// Mitsubishi GX Works2 project: wakom   PLC: Q02/Q02H

TYPE QD75_POS : STRUCT
  id : INT;
  mcode : INT;
  dwell_time : INT;
  spare : INT;
  speed : DINT;
  address : DINT;
  arc_address : DINT;
END_STRUCT END_TYPE

TYPE CAR_DATA : STRUCT
  cid : INT;
  enter_time : ARRAY [0..6] OF INT;
  leave_time : ARRAY [0..6] OF INT;
  proc_time : ARRAY [0..6] OF INT;
END_STRUCT END_TYPE

TYPE TK_POS : STRUCT
  h_lock : DINT;
  h_unlock : DINT;
  v_bottom : DINT;
  h_lock2 : DINT;
  h_unlock2 : DINT;
  v_bottom2 : DINT;
END_STRUCT END_TYPE

TYPE TK_CNF : STRUCT
  take_weight : INT;
  next_tank : ARRAY [0..4] OF INT;
  is_bypass : INT;
END_STRUCT END_TYPE

TYPE RECIPE : STRUCT
  tk_data : ARRAY [0..249] OF INT;
  sys_data : INT;
END_STRUCT END_TYPE

TYPE TK_STATUS : STRUCT
  permit_put : BOOL;
  cover_is_open : BOOL;
  cmd_open_cover : BOOL;
  cmd_close_cover : BOOL;
  permit_take : BOOL;
  rb_inter_lock : INT;
  pc_key : INT;
END_STRUCT END_TYPE

TYPE RB_STATUS : STRUCT
  pc_tid : INT;
  pc_key : INT;
  h_cur_pos : DINT;
  v_cur_pos : DINT;
  v_error_code : INT;
  v_alarm_code : INT;
  v_serve_alarm_code : INT;
  v_action_status : INT;
  v_status : INT;
  rb_state : INT;
  target_tid : INT;
  cur_tid : INT;
  from_tid : INT;
  to_tid : INT;
  v_xy : INT;
  v_cur_speed : DINT;
  v_bit : INT;
  h_cur_speed : DINT;
  h_error_code : INT;
  h_alarm_code : INT;
  h_serve_alarm_code : INT;
  h_action_status : INT;
  h_status : INT;
  h_xy : INT;
  h_bit : INT;
  h_address : DINT;
  h_speed : DINT;
  v_address : DINT;
  v_speed : DINT;
  rb_bit : INT;
END_STRUCT END_TYPE

TYPE SYS_STATUS : STRUCT
  amode : BOOL;
  mmode : BOOL;
  cycle_stop : BOOL;
  enable_run : BOOL;
  key_reset : BOOL;
  rcpid : INT;
END_STRUCT END_TYPE

TYPE ALARM : STRUCT
  tk : ARRAY [0..6] OF DINT;
  rb : ARRAY [0..0] OF DINT;
  emo : BOOL;
  leak : BOOL;
END_STRUCT END_TYPE

TYPE DIW_RCP : STRUCT
  LoopCount : INT;
  uiRemain : ARRAY [0..5] OF INT;
  uiCmd : ARRAY [0..5] OF INT;
  spare : ARRAY [0..36] OF INT;
END_STRUCT END_TYPE

// global labels: Global1
VAR_GLOBAL
  g_tk_status : ARRAY [0..6] OF TK_STATUS;
  g_rb_status : ARRAY [0..0] OF RB_STATUS;
  g_pc_cmd AT D900 : ARRAY [0..99] OF INT;
  g_recipe : RECIPE;
  g_tk_cnf : ARRAY [0..6] OF TK_CNF;
  g_tk_pos : ARRAY [0..6] OF TK_POS;
END_VAR
VAR_GLOBAL CONSTANT
  g_safe_height : DINT;
END_VAR
VAR_GLOBAL
  g_tk_car : ARRAY [0..6] OF CAR_DATA;
  g_rb_car : ARRAY [0..0] OF CAR_DATA;
  g_sys_status : SYS_STATUS;
  g_alarm : ALARM;
END_VAR
VAR_GLOBAL CONSTANT
  g_rcp_max_size : INT := 50;
END_VAR

// task task01 (event TRUE, interval 0, priority 31): robot01
// task task02 (event TRUE, interval 0, priority 31): main

PROGRAM robot01
VAR
  axis_h : rb_axis;
  axis_v : rb_axis;
  rb_dispatch_1 : rb_dispatch;
END_VAR
(* structured ladder/FBD written out as ST: instructions are called as NAME(EN, inputs, outputs); _pN, _eN, _tN stand for wires *)
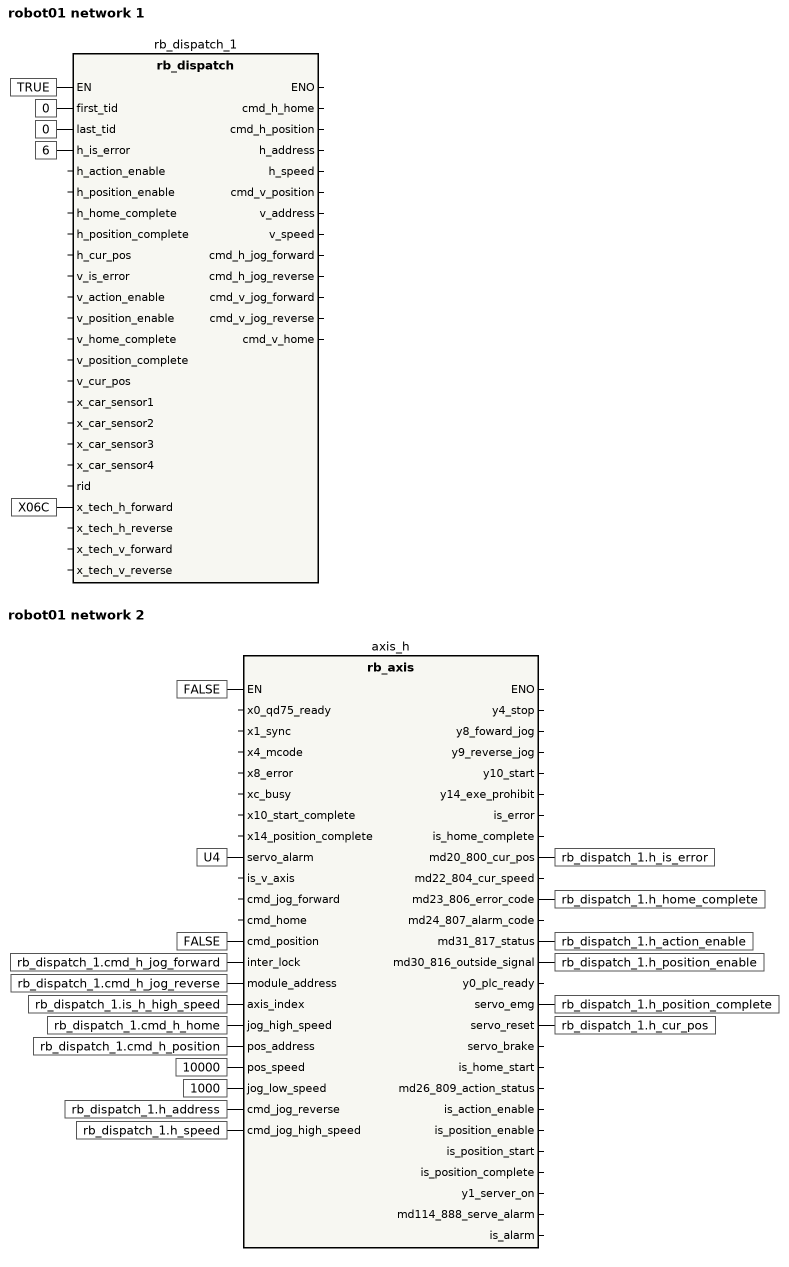
(* network 1 *)
rb_dispatch_1(EN := TRUE, first_tid := 0, last_tid := 0, h_is_error := 6, x_tech_h_forward := X06C);
(* network 2 *)
axis_h(EN := FALSE, servo_alarm := U4, cmd_position := FALSE, inter_lock := rb_dispatch_1.cmd_h_jog_forward, module_address := rb_dispatch_1.cmd_h_jog_reverse, axis_index := rb_dispatch_1.is_h_high_speed, jog_high_speed := rb_dispatch_1.cmd_h_home, pos_address := rb_dispatch_1.cmd_h_position, pos_speed := 10000, jog_low_speed := 1000, cmd_jog_reverse := rb_dispatch_1.h_address, cmd_jog_high_speed := rb_dispatch_1.h_speed, md20_800_cur_pos => rb_dispatch_1.h_is_error, md23_806_error_code => rb_dispatch_1.h_home_complete, md31_817_status => rb_dispatch_1.h_action_enable, md30_816_outside_signal => rb_dispatch_1.h_position_enable, servo_emg => rb_dispatch_1.h_position_complete, servo_reset => rb_dispatch_1.h_cur_pos);
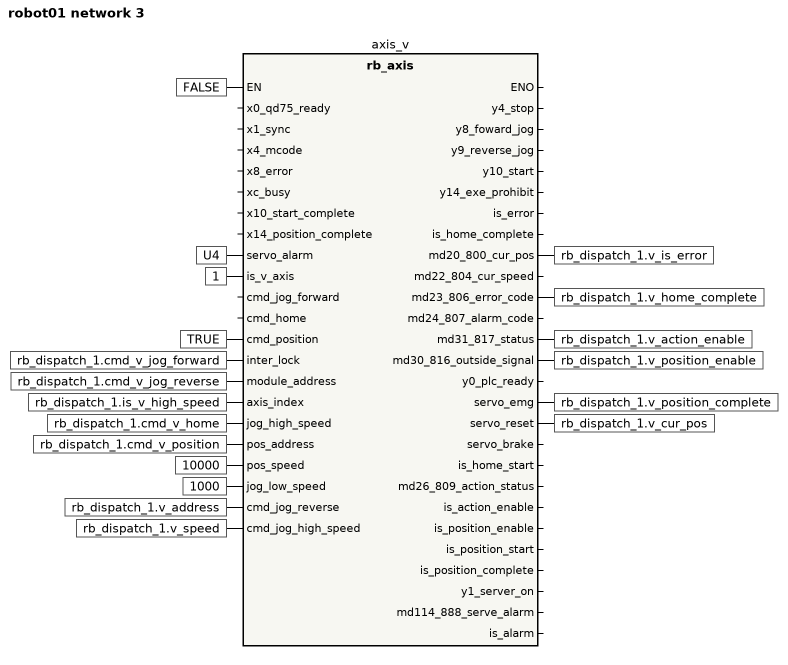
(* network 3 *)
axis_v(EN := FALSE, servo_alarm := U4, is_v_axis := 1, cmd_position := TRUE, inter_lock := rb_dispatch_1.cmd_v_jog_forward, module_address := rb_dispatch_1.cmd_v_jog_reverse, axis_index := rb_dispatch_1.is_v_high_speed, jog_high_speed := rb_dispatch_1.cmd_v_home, pos_address := rb_dispatch_1.cmd_v_position, pos_speed := 10000, jog_low_speed := 1000, cmd_jog_reverse := rb_dispatch_1.v_address, cmd_jog_high_speed := rb_dispatch_1.v_speed, md20_800_cur_pos => rb_dispatch_1.v_is_error, md23_806_error_code => rb_dispatch_1.v_home_complete, md31_817_status => rb_dispatch_1.v_action_enable, md30_816_outside_signal => rb_dispatch_1.v_position_enable, servo_emg => rb_dispatch_1.v_position_complete, servo_reset => rb_dispatch_1.v_cur_pos);
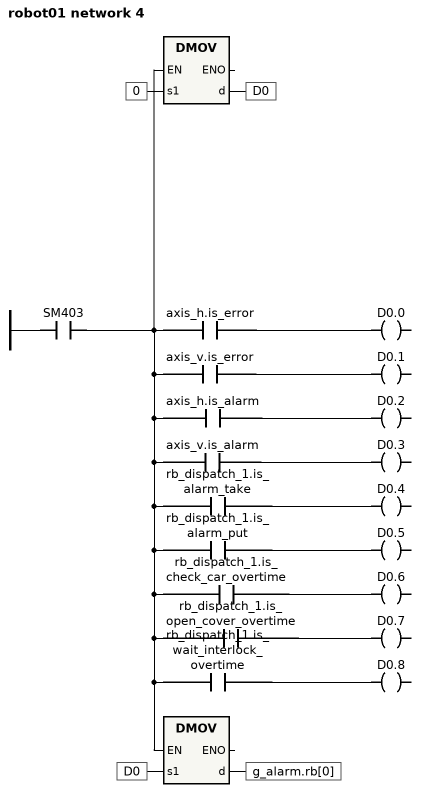
(* network 4 *)
DMOV(SM403, 0, D0);
D0.0 := SM403 AND axis_h.is_error;
D0.1 := SM403 AND axis_v.is_error;
D0.2 := SM403 AND axis_h.is_alarm;
D0.3 := SM403 AND axis_v.is_alarm;
D0.4 := SM403 AND rb_dispatch_1.is_alarm_take;
D0.5 := SM403 AND rb_dispatch_1.is_alarm_put;
D0.6 := SM403 AND rb_dispatch_1.is_check_car_overtime;
D0.7 := SM403 AND rb_dispatch_1.is_open_cover_overtime;
D0.8 := SM403 AND rb_dispatch_1.is_wait_interlock_overtime;
DMOV(SM403, D0, g_alarm.rb[0]);
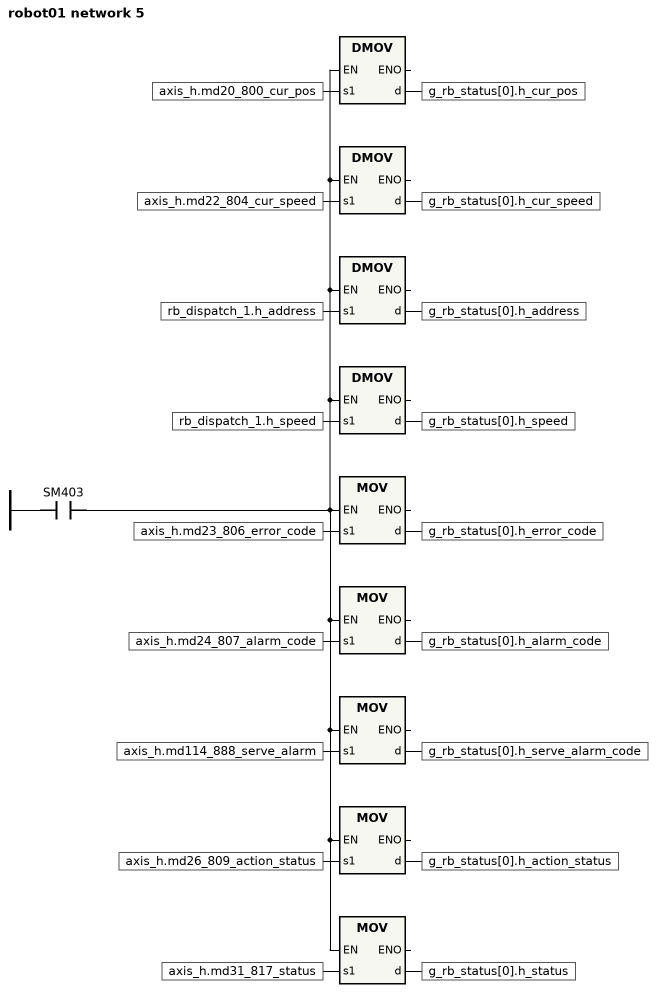
(* network 5 *)
DMOV(SM403, axis_h.md20_800_cur_pos, g_rb_status[0].h_cur_pos);
DMOV(SM403, axis_h.md22_804_cur_speed, g_rb_status[0].h_cur_speed);
DMOV(SM403, rb_dispatch_1.h_address, g_rb_status[0].h_address);
DMOV(SM403, rb_dispatch_1.h_speed, g_rb_status[0].h_speed);
MOV(SM403, axis_h.md23_806_error_code, g_rb_status[0].h_error_code);
MOV(SM403, axis_h.md24_807_alarm_code, g_rb_status[0].h_alarm_code);
MOV(SM403, axis_h.md114_888_serve_alarm, g_rb_status[0].h_serve_alarm_code);
MOV(SM403, axis_h.md26_809_action_status, g_rb_status[0].h_action_status);
MOV(SM403, axis_h.md31_817_status, g_rb_status[0].h_status);
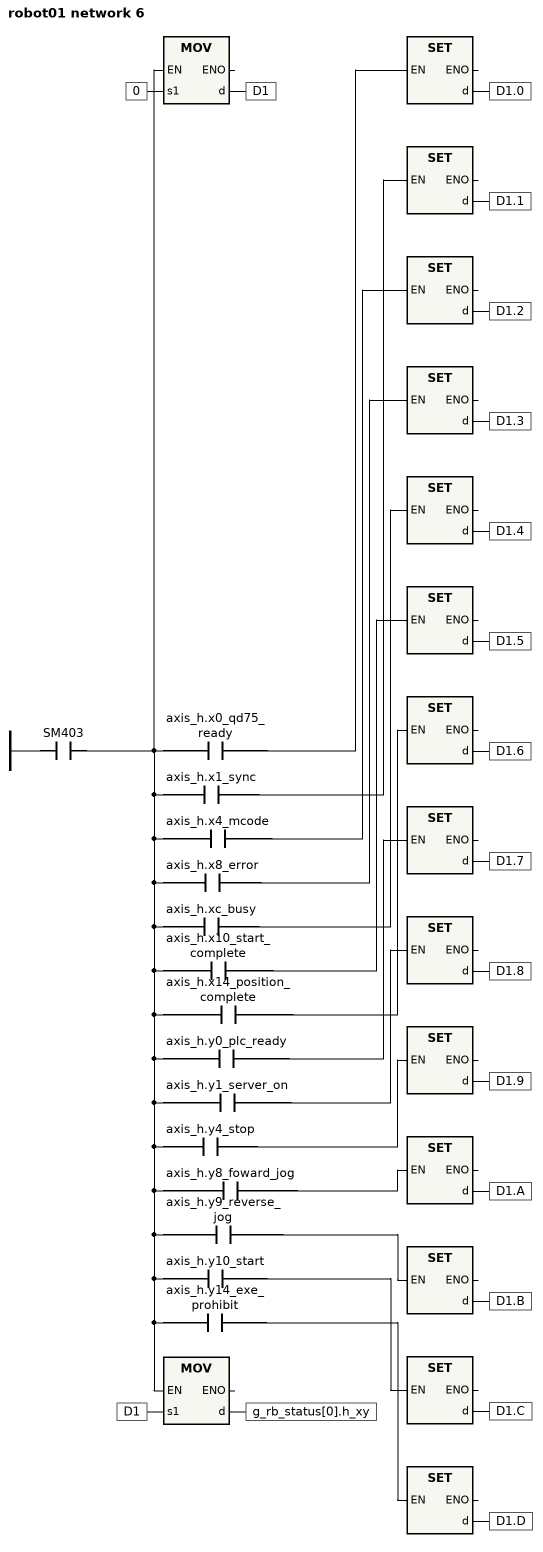
(* network 6 *)
MOV(SM403, 0, D1);
SET(SM403 AND axis_h.x0_qd75_ready, D1.0);
SET(SM403 AND axis_h.x1_sync, D1.1);
SET(SM403 AND axis_h.x4_mcode, D1.2);
SET(SM403 AND axis_h.x8_error, D1.3);
SET(SM403 AND axis_h.xc_busy, D1.4);
SET(SM403 AND axis_h.x10_start_complete, D1.5);
SET(SM403 AND axis_h.x14_position_complete, D1.6);
SET(SM403 AND axis_h.y0_plc_ready, D1.7);
SET(SM403 AND axis_h.y1_server_on, D1.8);
SET(SM403 AND axis_h.y4_stop, D1.9);
SET(SM403 AND axis_h.y8_foward_jog, D1.A);
SET(SM403 AND axis_h.y9_reverse_jog, D1.B);
SET(SM403 AND axis_h.y10_start, D1.C);
SET(SM403 AND axis_h.y14_exe_prohibit, D1.D);
MOV(SM403, D1, g_rb_status[0].h_xy);
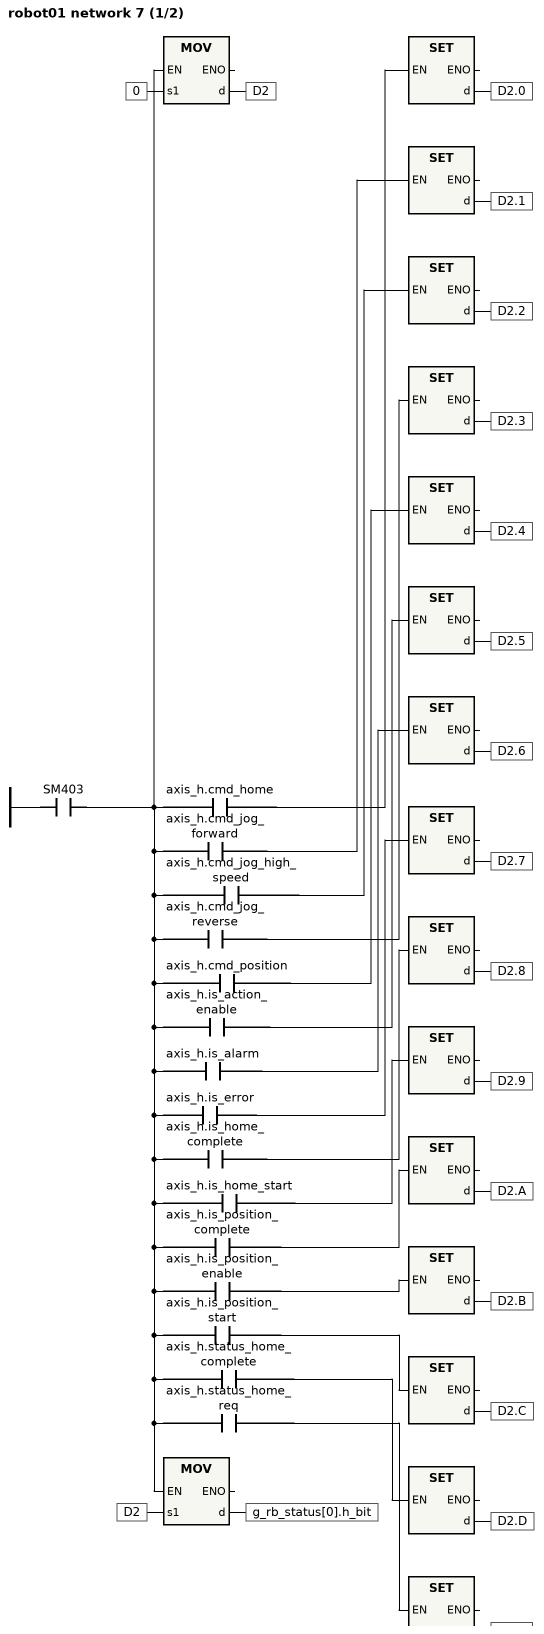
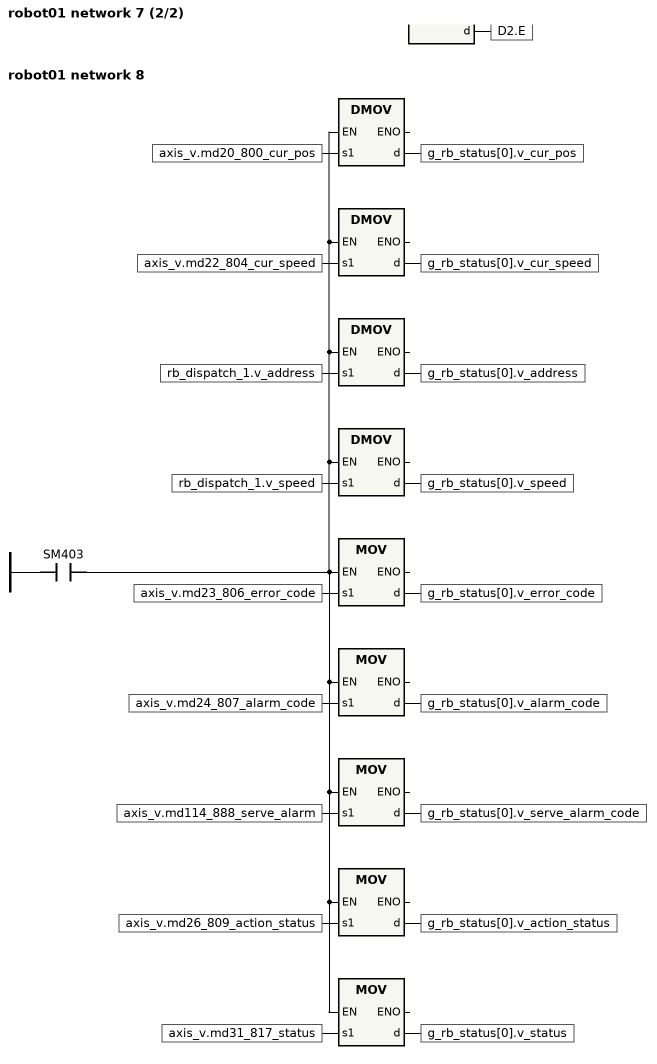
(* network 7 *)
MOV(SM403, 0, D2);
SET(SM403 AND axis_h.cmd_home, D2.0);
SET(SM403 AND axis_h.cmd_jog_forward, D2.1);
SET(SM403 AND axis_h.cmd_jog_high_speed, D2.2);
SET(SM403 AND axis_h.cmd_jog_reverse, D2.3);
SET(SM403 AND axis_h.cmd_position, D2.4);
SET(SM403 AND axis_h.is_action_enable, D2.5);
SET(SM403 AND axis_h.is_alarm, D2.6);
SET(SM403 AND axis_h.is_error, D2.7);
SET(SM403 AND axis_h.is_home_complete, D2.8);
SET(SM403 AND axis_h.is_home_start, D2.9);
SET(SM403 AND axis_h.is_position_complete, D2.A);
SET(SM403 AND axis_h.is_position_enable, D2.B);
SET(SM403 AND axis_h.is_position_start, D2.C);
SET(SM403 AND axis_h.status_home_complete, D2.D);
SET(SM403 AND axis_h.status_home_req, D2.E);
MOV(SM403, D2, g_rb_status[0].h_bit);
(* network 8 *)
DMOV(SM403, axis_v.md20_800_cur_pos, g_rb_status[0].v_cur_pos);
DMOV(SM403, axis_v.md22_804_cur_speed, g_rb_status[0].v_cur_speed);
DMOV(SM403, rb_dispatch_1.v_address, g_rb_status[0].v_address);
DMOV(SM403, rb_dispatch_1.v_speed, g_rb_status[0].v_speed);
MOV(SM403, axis_v.md23_806_error_code, g_rb_status[0].v_error_code);
MOV(SM403, axis_v.md24_807_alarm_code, g_rb_status[0].v_alarm_code);
MOV(SM403, axis_v.md114_888_serve_alarm, g_rb_status[0].v_serve_alarm_code);
MOV(SM403, axis_v.md26_809_action_status, g_rb_status[0].v_action_status);
MOV(SM403, axis_v.md31_817_status, g_rb_status[0].v_status);
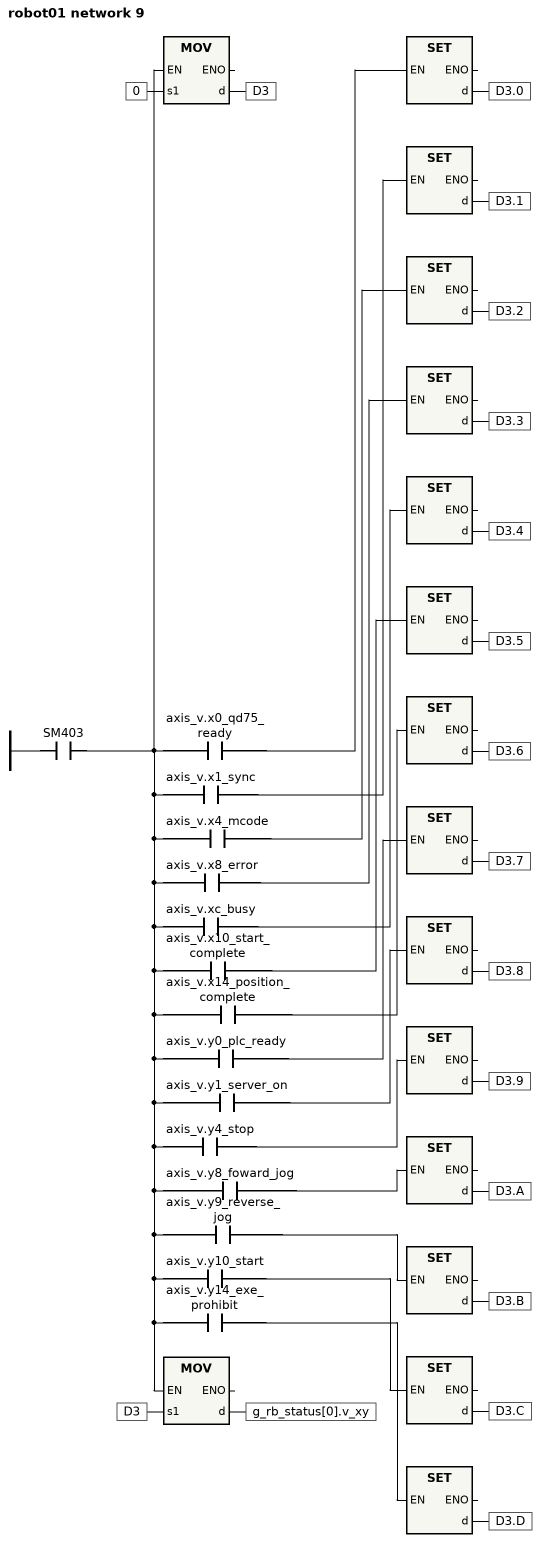
(* network 9 *)
MOV(SM403, 0, D3);
SET(SM403 AND axis_v.x0_qd75_ready, D3.0);
SET(SM403 AND axis_v.x1_sync, D3.1);
SET(SM403 AND axis_v.x4_mcode, D3.2);
SET(SM403 AND axis_v.x8_error, D3.3);
SET(SM403 AND axis_v.xc_busy, D3.4);
SET(SM403 AND axis_v.x10_start_complete, D3.5);
SET(SM403 AND axis_v.x14_position_complete, D3.6);
SET(SM403 AND axis_v.y0_plc_ready, D3.7);
SET(SM403 AND axis_v.y1_server_on, D3.8);
SET(SM403 AND axis_v.y4_stop, D3.9);
SET(SM403 AND axis_v.y8_foward_jog, D3.A);
SET(SM403 AND axis_v.y9_reverse_jog, D3.B);
SET(SM403 AND axis_v.y10_start, D3.C);
SET(SM403 AND axis_v.y14_exe_prohibit, D3.D);
MOV(SM403, D3, g_rb_status[0].v_xy);
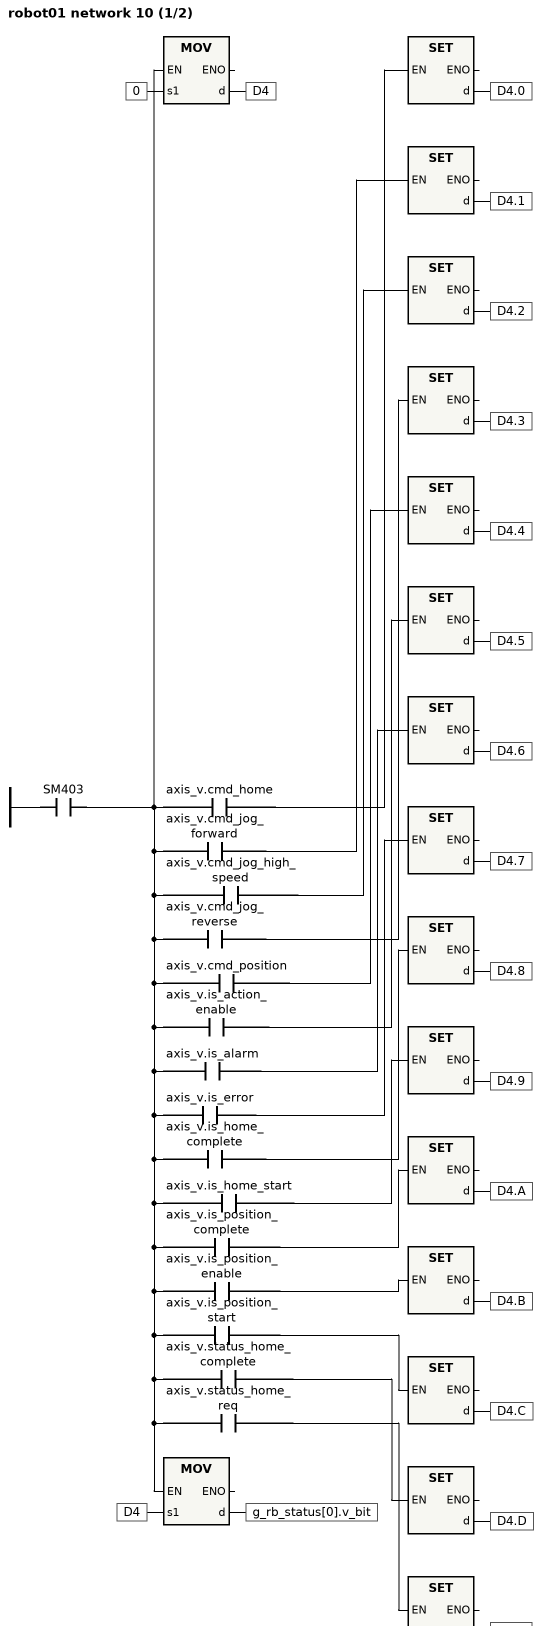
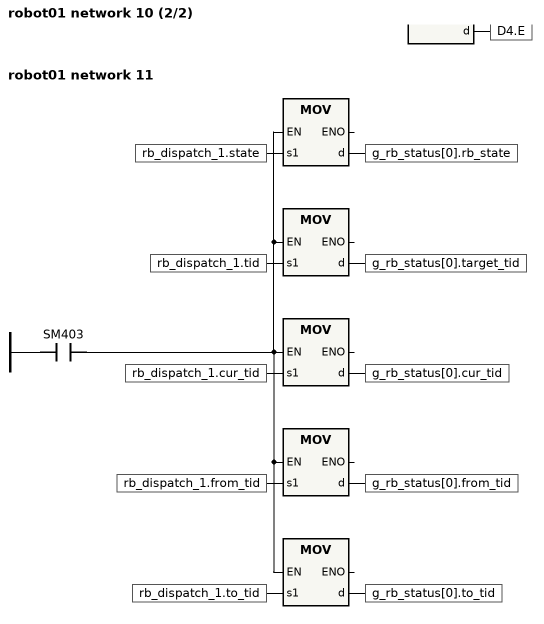
(* network 10 *)
MOV(SM403, 0, D4);
SET(SM403 AND axis_v.cmd_home, D4.0);
SET(SM403 AND axis_v.cmd_jog_forward, D4.1);
SET(SM403 AND axis_v.cmd_jog_high_speed, D4.2);
SET(SM403 AND axis_v.cmd_jog_reverse, D4.3);
SET(SM403 AND axis_v.cmd_position, D4.4);
SET(SM403 AND axis_v.is_action_enable, D4.5);
SET(SM403 AND axis_v.is_alarm, D4.6);
SET(SM403 AND axis_v.is_error, D4.7);
SET(SM403 AND axis_v.is_home_complete, D4.8);
SET(SM403 AND axis_v.is_home_start, D4.9);
SET(SM403 AND axis_v.is_position_complete, D4.A);
SET(SM403 AND axis_v.is_position_enable, D4.B);
SET(SM403 AND axis_v.is_position_start, D4.C);
SET(SM403 AND axis_v.status_home_complete, D4.D);
SET(SM403 AND axis_v.status_home_req, D4.E);
MOV(SM403, D4, g_rb_status[0].v_bit);
(* network 11 *)
MOV(SM403, rb_dispatch_1.state, g_rb_status[0].rb_state);
MOV(SM403, rb_dispatch_1.tid, g_rb_status[0].target_tid);
MOV(SM403, rb_dispatch_1.cur_tid, g_rb_status[0].cur_tid);
MOV(SM403, rb_dispatch_1.from_tid, g_rb_status[0].from_tid);
MOV(SM403, rb_dispatch_1.to_tid, g_rb_status[0].to_tid);
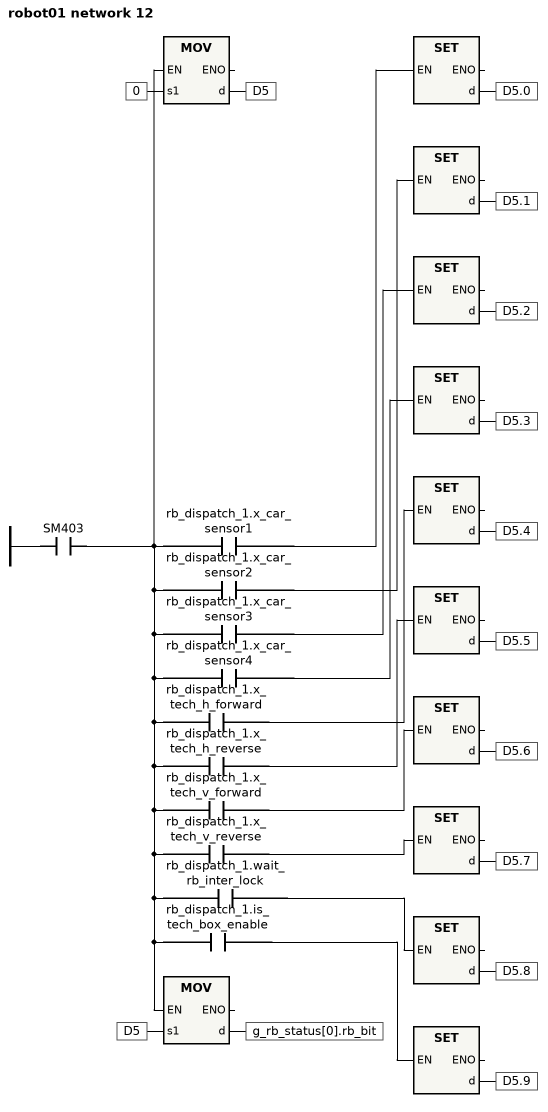
(* network 12 *)
MOV(SM403, 0, D5);
SET(SM403 AND rb_dispatch_1.x_car_sensor1, D5.0);
SET(SM403 AND rb_dispatch_1.x_car_sensor2, D5.1);
SET(SM403 AND rb_dispatch_1.x_car_sensor3, D5.2);
SET(SM403 AND rb_dispatch_1.x_car_sensor4, D5.3);
SET(SM403 AND rb_dispatch_1.x_tech_h_forward, D5.4);
SET(SM403 AND rb_dispatch_1.x_tech_h_reverse, D5.5);
SET(SM403 AND rb_dispatch_1.x_tech_v_forward, D5.6);
SET(SM403 AND rb_dispatch_1.x_tech_v_reverse, D5.7);
SET(SM403 AND rb_dispatch_1.wait_rb_inter_lock, D5.8);
SET(SM403 AND rb_dispatch_1.is_tech_box_enable, D5.9);
MOV(SM403, D5, g_rb_status[0].rb_bit);
END_PROGRAM

FUNCTION_BLOCK rb_axis
VAR_INPUT
  x0_qd75_ready : BOOL;
  x1_sync : BOOL;
  x4_mcode : BOOL;
  x8_error : BOOL;
  xc_busy : BOOL;
  x10_start_complete : BOOL;
END_VAR
VAR_OUTPUT
  y4_stop : BOOL;
  y8_foward_jog : BOOL;
  y9_reverse_jog : BOOL;
  y10_start : BOOL;  (* 定位启动信号 *)
END_VAR
VAR_INPUT
  x14_position_complete : BOOL;
END_VAR
VAR_OUTPUT
  y14_exe_prohibit : BOOL;
  is_error : BOOL;
  is_home_complete : BOOL;
END_VAR
VAR CONSTANT
  cd5_1502_error_reset : INT := 1502;
  cd7_1504_mcode_off : INT := 1504;
END_VAR
VAR_OUTPUT
  md20_800_cur_pos : DINT;
  md22_804_cur_speed : DINT;
  md23_806_error_code : INT;
  md24_807_alarm_code : INT;
  md31_817_status : INT;
  md30_816_outside_signal : WORD;  (* Md.30外部输入输出信号 *)
  y0_plc_ready : BOOL;
  servo_emg : BOOL;
  servo_reset : BOOL;
  servo_brake : BOOL;
END_VAR
VAR_INPUT
  servo_alarm : BOOL;
  is_v_axis : BOOL;
  cmd_jog_forward : BOOL;
END_VAR
VAR CONSTANT
  cd17_1518_jog_speed : INT := 1518;
END_VAR
VAR_INPUT
  cmd_home : BOOL;
END_VAR
VAR_OUTPUT
  is_home_start : BOOL;
END_VAR
VAR_INPUT
  cmd_position : BOOL;
END_VAR
VAR CONSTANT
  cd3_1500_position_num : INT := 1500;
  da2000_position : INT := 2000;
END_VAR
VAR_OUTPUT
  md26_809_action_status : INT;
  is_action_enable : BOOL;
  is_position_enable : BOOL;
  is_position_start : BOOL;
  is_position_complete : BOOL;
END_VAR
VAR_INPUT
  inter_lock : BOOL;
  module_address : INT;
  axis_index : INT;
  jog_high_speed : DINT;
  pos_address : DINT;
END_VAR
VAR
  outside_down_limit : BOOL;
  outside_up_limit : BOOL;
  outside_stop : BOOL;
  status_home_req : BOOL;
  status_home_complete : BOOL;
END_VAR
VAR_INPUT
  pos_speed : DINT;
END_VAR
VAR
  pos_data : QD75_POS;
  home_overtime : BOOL;
  TON_home : TON;
END_VAR
VAR CONSTANT
  TON_home_time : TIME;
END_VAR
VAR
  position_overtime : BOOL;
  TON_position : TON;
END_VAR
VAR CONSTANT
  TON_position_time : TIME;
END_VAR
VAR_INPUT
  jog_low_speed : DINT;
END_VAR
VAR_OUTPUT
  y1_server_on : BOOL;
END_VAR
VAR_INPUT
  cmd_jog_reverse : BOOL;
  cmd_jog_high_speed : BOOL;
END_VAR
VAR_OUTPUT
  md114_888_serve_alarm : INT;
  is_alarm : BOOL;
END_VAR
VAR
  status_alarm : BOOL;
END_VAR
(* structured ladder/FBD written out as ST: instructions are called as NAME(EN, inputs, outputs); _pN, _eN, _tN stand for wires *)
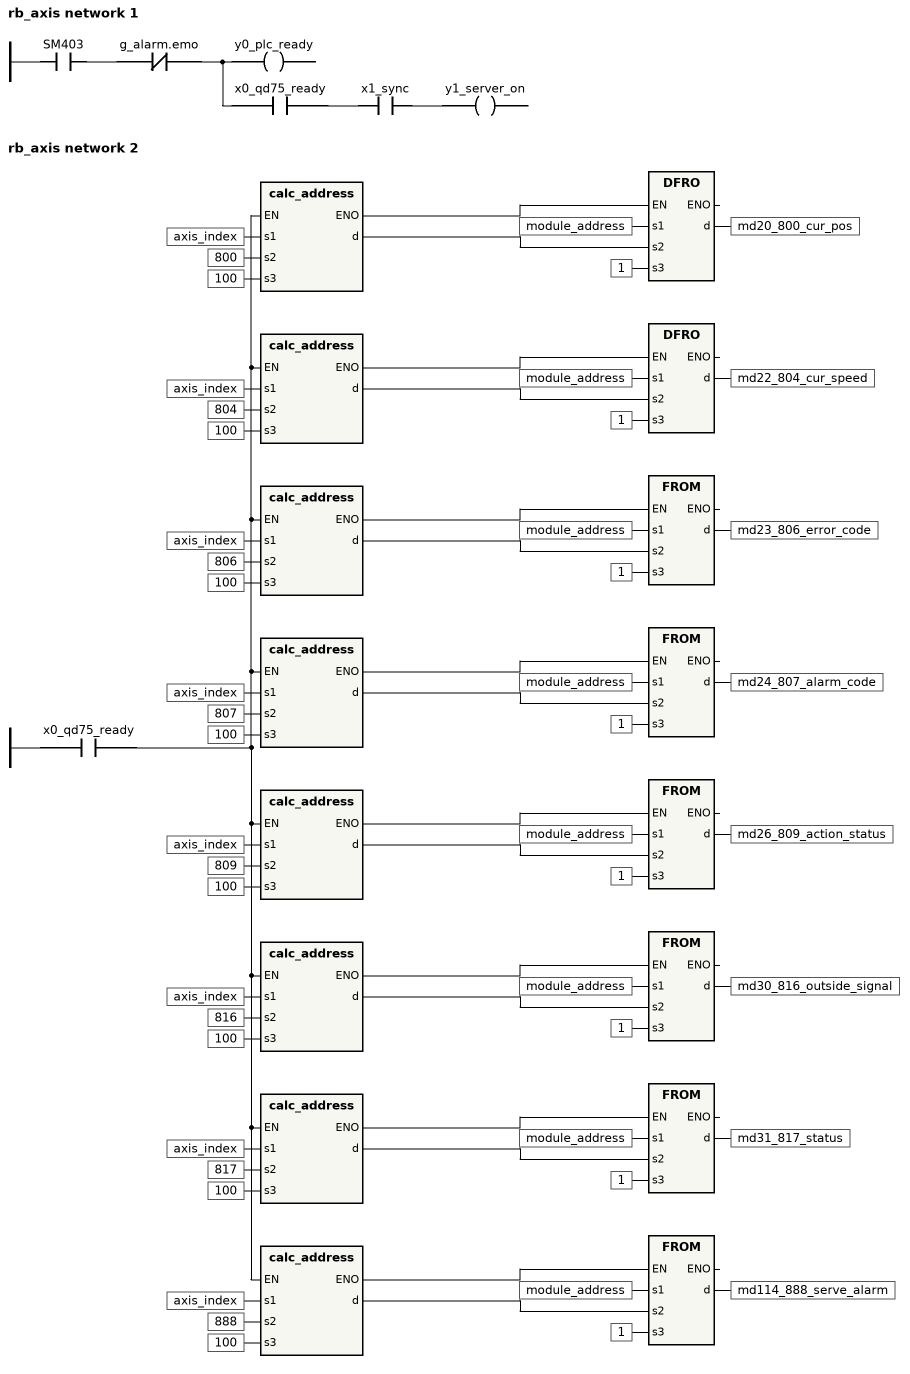
(* network 1 *)
_p1 := SM403 AND NOT g_alarm.emo;
y0_plc_ready := _p1;
y1_server_on := _p1 AND x0_qd75_ready AND x1_sync;
(* network 2 *)
_e2 := calc_address(x0_qd75_ready, axis_index, 800, 100, _t1);
DFRO(_e2, module_address, _t1, 1, md20_800_cur_pos);
_e4 := calc_address(x0_qd75_ready, axis_index, 804, 100, _t3);
DFRO(_e4, module_address, _t3, 1, md22_804_cur_speed);
_e6 := calc_address(x0_qd75_ready, axis_index, 806, 100, _t5);
FROM(_e6, module_address, _t5, 1, md23_806_error_code);
_e8 := calc_address(x0_qd75_ready, axis_index, 807, 100, _t7);
FROM(_e8, module_address, _t7, 1, md24_807_alarm_code);
_e10 := calc_address(x0_qd75_ready, axis_index, 809, 100, _t9);
FROM(_e10, module_address, _t9, 1, md26_809_action_status);
_e12 := calc_address(x0_qd75_ready, axis_index, 816, 100, _t11);
FROM(_e12, module_address, _t11, 1, md30_816_outside_signal);
_e14 := calc_address(x0_qd75_ready, axis_index, 817, 100, _t13);
FROM(_e14, module_address, _t13, 1, md31_817_status);
_e16 := calc_address(x0_qd75_ready, axis_index, 888, 100, _t15);
FROM(_e16, module_address, _t15, 1, md114_888_serve_alarm);
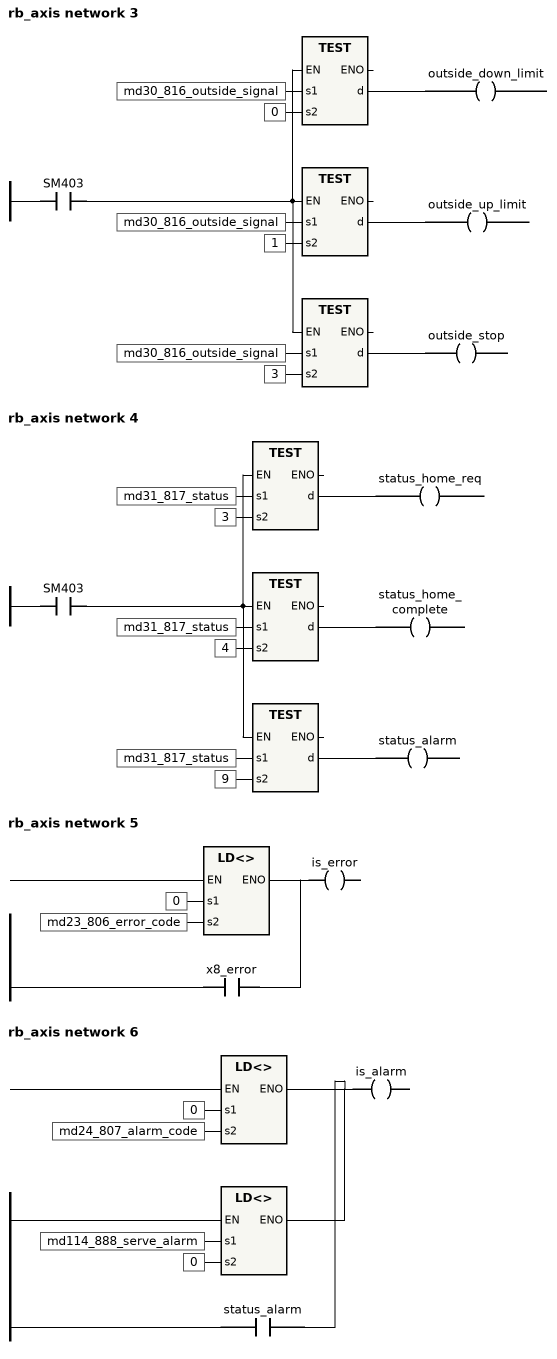
(* network 3 *)
TEST(SM403, md30_816_outside_signal, 0, _t1);
outside_down_limit := _t1;
TEST(SM403, md30_816_outside_signal, 1, _t2);
outside_up_limit := _t2;
TEST(SM403, md30_816_outside_signal, 3, _t3);
outside_stop := _t3;
(* network 4 *)
TEST(SM403, md31_817_status, 3, _t1);
status_home_req := _t1;
TEST(SM403, md31_817_status, 4, _t2);
status_home_complete := _t2;
TEST(SM403, md31_817_status, 9, _t3);
status_alarm := _t3;
(* network 5 *)
_e1 := LD<>(TRUE, 0, md23_806_error_code);
is_error := _e1 OR x8_error;
(* network 6 *)
_e1 := LD<>(TRUE, 0, md24_807_alarm_code);
_e2 := LD<>(TRUE, md114_888_serve_alarm, 0);
is_alarm := _e1 OR status_alarm OR _e2;
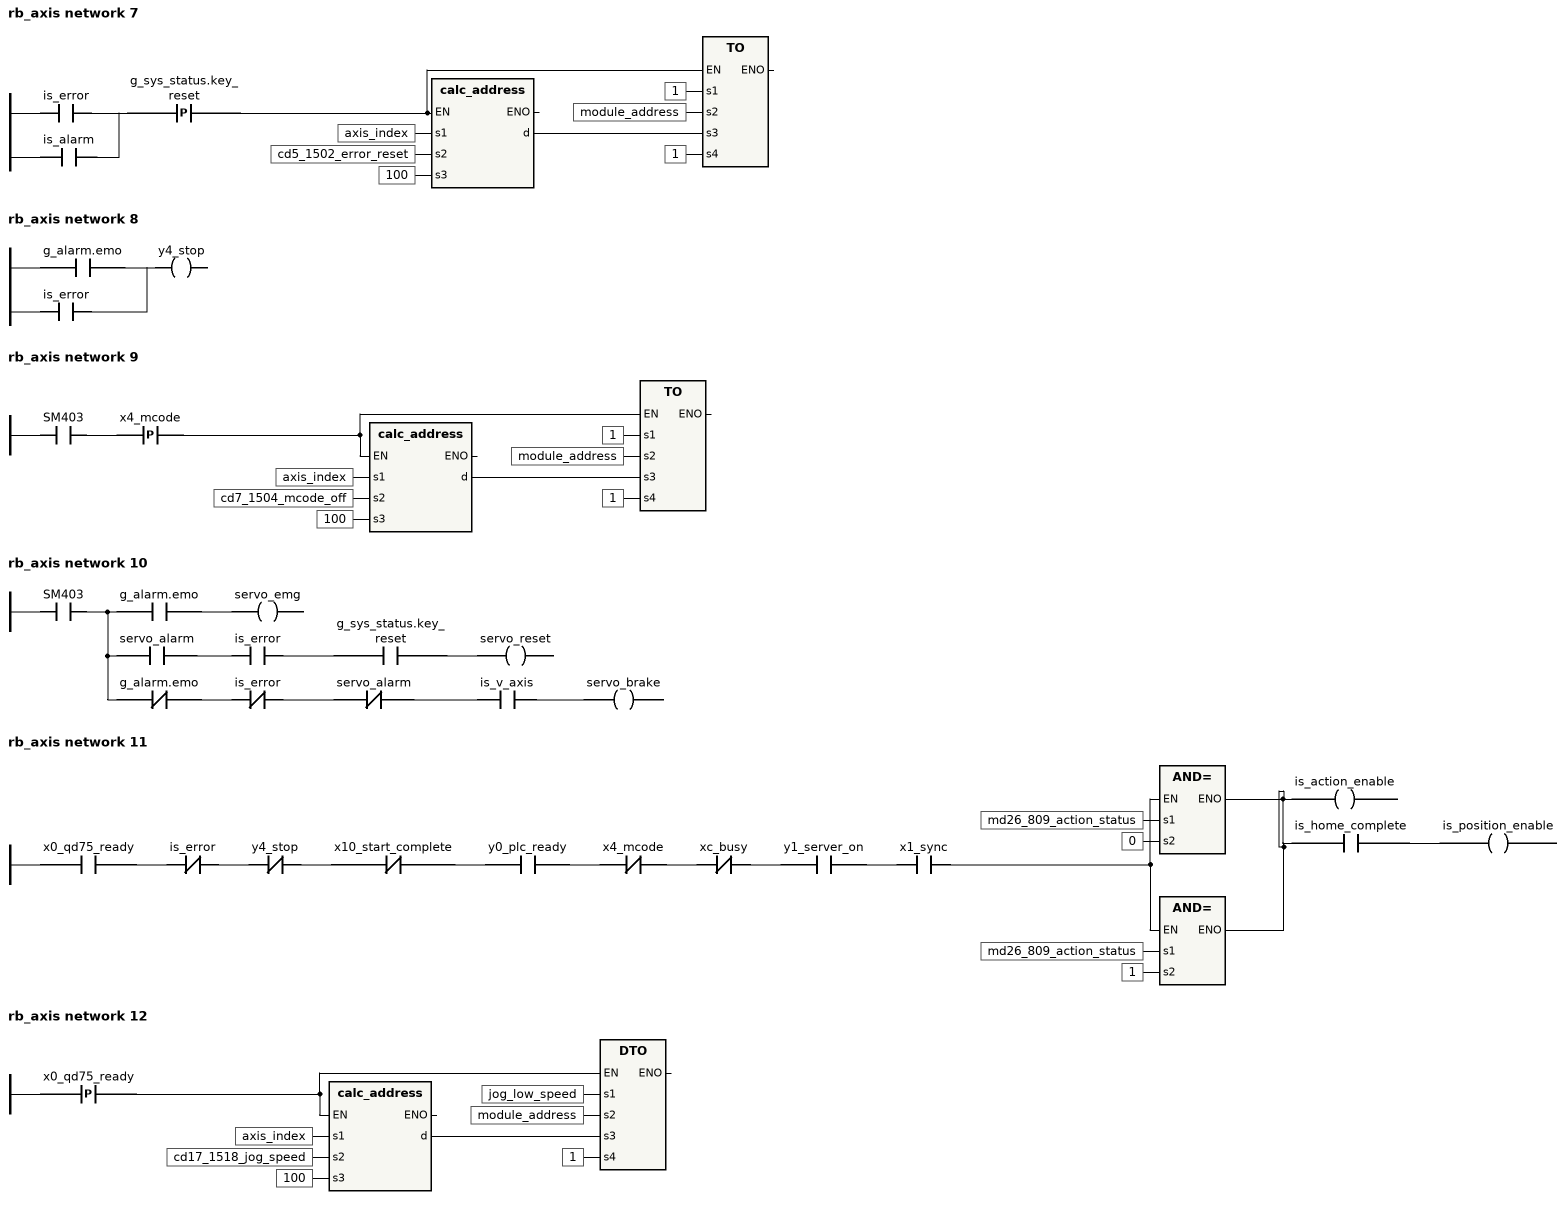
(* network 7 *)
_p1 := (is_error OR is_alarm) AND LDP(TRUE, g_sys_status.key_reset);
calc_address(_p1, axis_index, cd5_1502_error_reset, 100, _t2);
TO(_p1, 1, module_address, _t2, 1);
(* network 8 *)
y4_stop := g_alarm.emo OR is_error;
(* network 9 *)
_p1 := SM403 AND LDP(TRUE, x4_mcode);
calc_address(_p1, axis_index, cd7_1504_mcode_off, 100, _t2);
TO(_p1, 1, module_address, _t2, 1);
(* network 10 *)
servo_emg := SM403 AND g_alarm.emo;
servo_reset := SM403 AND servo_alarm AND is_error AND g_sys_status.key_reset;
servo_brake := SM403 AND NOT g_alarm.emo AND NOT is_error AND NOT servo_alarm AND is_v_axis;
(* network 11 *)
_p1 := x0_qd75_ready AND NOT is_error AND NOT y4_stop AND NOT x10_start_complete AND y0_plc_ready AND NOT x4_mcode AND NOT xc_busy AND y1_server_on AND x1_sync;
_e2 := AND=(_p1, md26_809_action_status, 0);
_e3 := AND=(_p1, md26_809_action_status, 1);
_p4 := _e2 OR _e3;
is_action_enable := _p4;
is_position_enable := _p4 AND is_home_complete;
(* network 12 *)
_p1 := LDP(TRUE, x0_qd75_ready);
calc_address(_p1, axis_index, cd17_1518_jog_speed, 100, _t2);
DTO(_p1, jog_low_speed, module_address, _t2, 1);
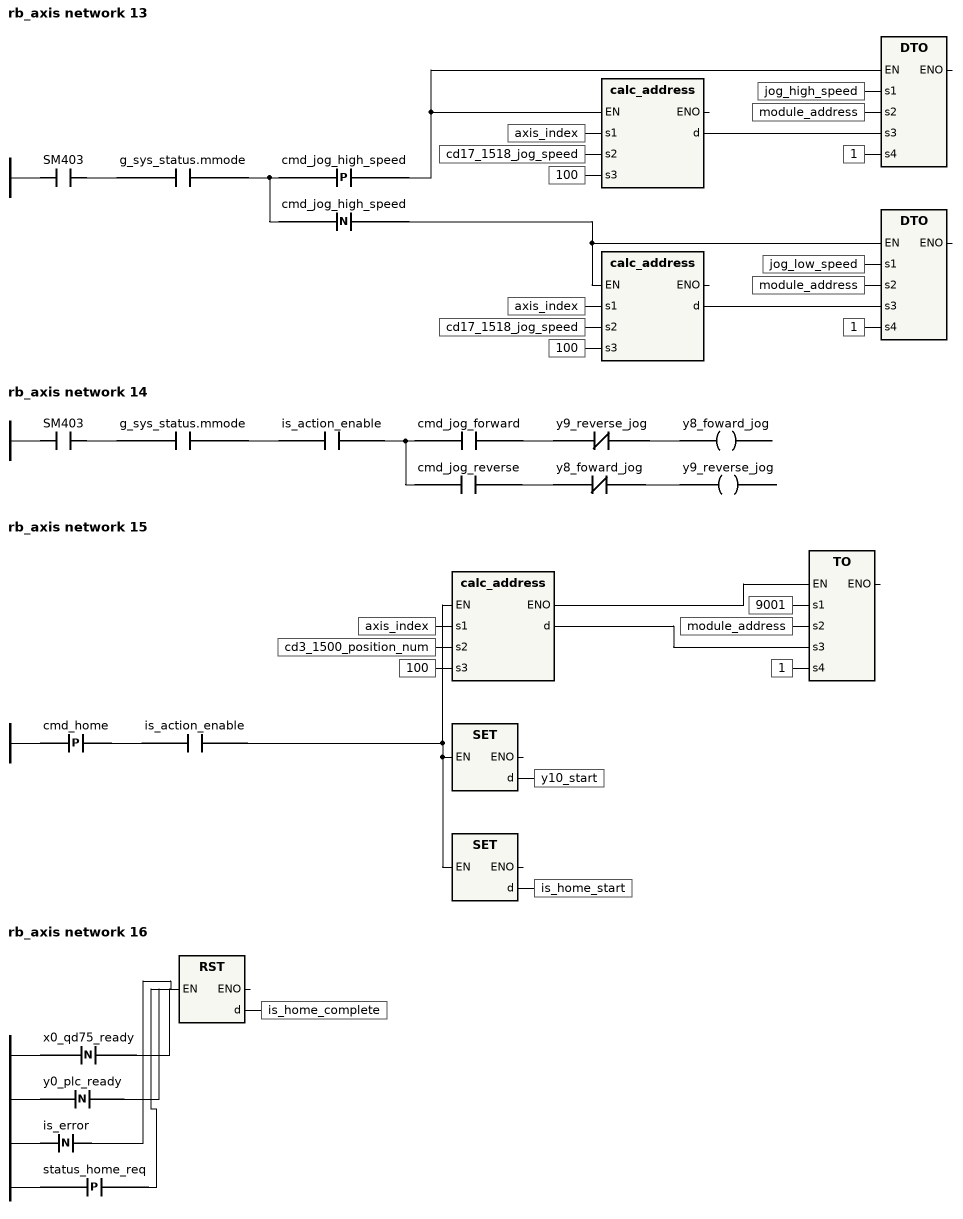
(* network 13 *)
_p1 := SM403 AND g_sys_status.mmode;
_p2 := _p1 AND LDP(TRUE, cmd_jog_high_speed);
calc_address(_p2, axis_index, cd17_1518_jog_speed, 100, _t3);
DTO(_p2, jog_high_speed, module_address, _t3, 1);
_p4 := _p1 AND LDF(TRUE, cmd_jog_high_speed);
calc_address(_p4, axis_index, cd17_1518_jog_speed, 100, _t5);
DTO(_p4, jog_low_speed, module_address, _t5, 1);
(* network 14 *)
_p1 := SM403 AND g_sys_status.mmode AND is_action_enable;
y8_foward_jog := _p1 AND cmd_jog_forward AND NOT y9_reverse_jog;
y9_reverse_jog := _p1 AND cmd_jog_reverse AND NOT y8_foward_jog;
(* network 15 *)
_p1 := LDP(TRUE, cmd_home) AND is_action_enable;
_e3 := calc_address(_p1, axis_index, cd3_1500_position_num, 100, _t2);
TO(_e3, 9001, module_address, _t2, 1);
SET(_p1, y10_start);
SET(_p1, is_home_start);
(* network 16 *)
RST(LDF(TRUE, x0_qd75_ready) OR LDF(TRUE, y0_plc_ready) OR LDF(TRUE, is_error) OR LDP(TRUE, status_home_req), is_home_complete);
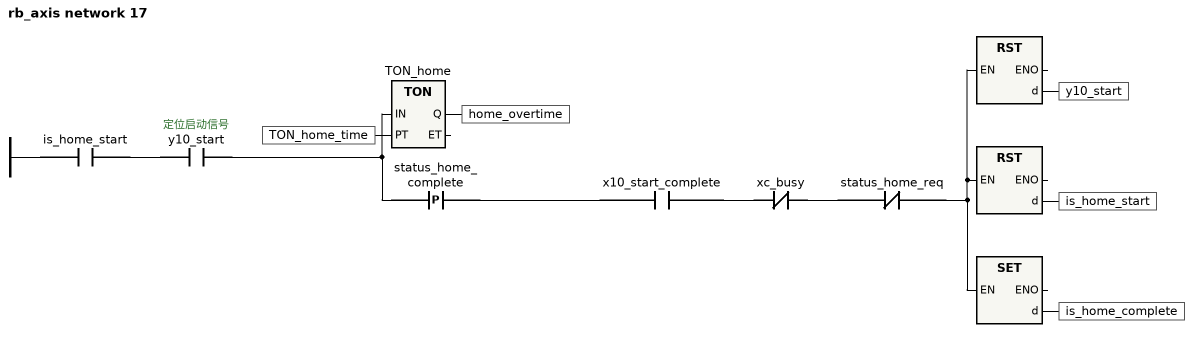
(* network 17 *)
_p1 := is_home_start AND y10_start;
_p2 := _p1 AND LDP(TRUE, status_home_complete) AND x10_start_complete AND NOT xc_busy AND NOT status_home_req;
RST(_p2, y10_start);
RST(_p2, is_home_start);
SET(_p2, is_home_complete);
TON_home(IN := _p1, PT := TON_home_time, Q => home_overtime);
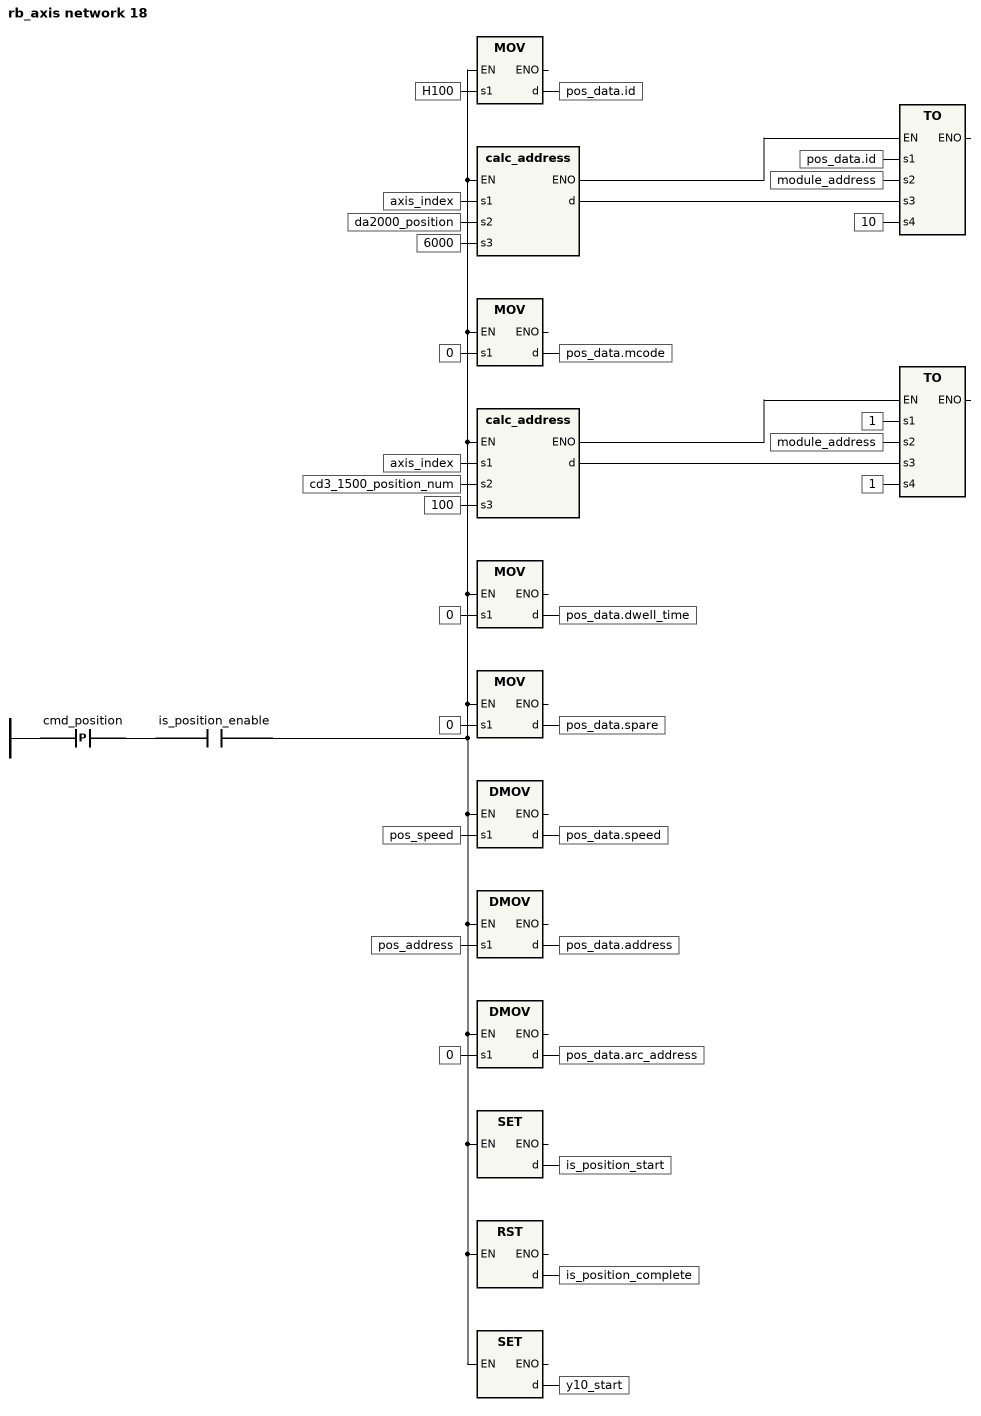
(* network 18 *)
_p1 := LDP(TRUE, cmd_position) AND is_position_enable;
MOV(_p1, H100, pos_data.id);
MOV(_p1, 0, pos_data.mcode);
MOV(_p1, 0, pos_data.dwell_time);
MOV(_p1, 0, pos_data.spare);
DMOV(_p1, pos_speed, pos_data.speed);
DMOV(_p1, pos_address, pos_data.address);
DMOV(_p1, 0, pos_data.arc_address);
_e3 := calc_address(_p1, axis_index, da2000_position, 6000, _t2);
TO(_e3, pos_data.id, module_address, _t2, 10);
_e5 := calc_address(_p1, axis_index, cd3_1500_position_num, 100, _t4);
TO(_e5, 1, module_address, _t4, 1);
SET(_p1, is_position_start);
RST(_p1, is_position_complete);
SET(_p1, y10_start);
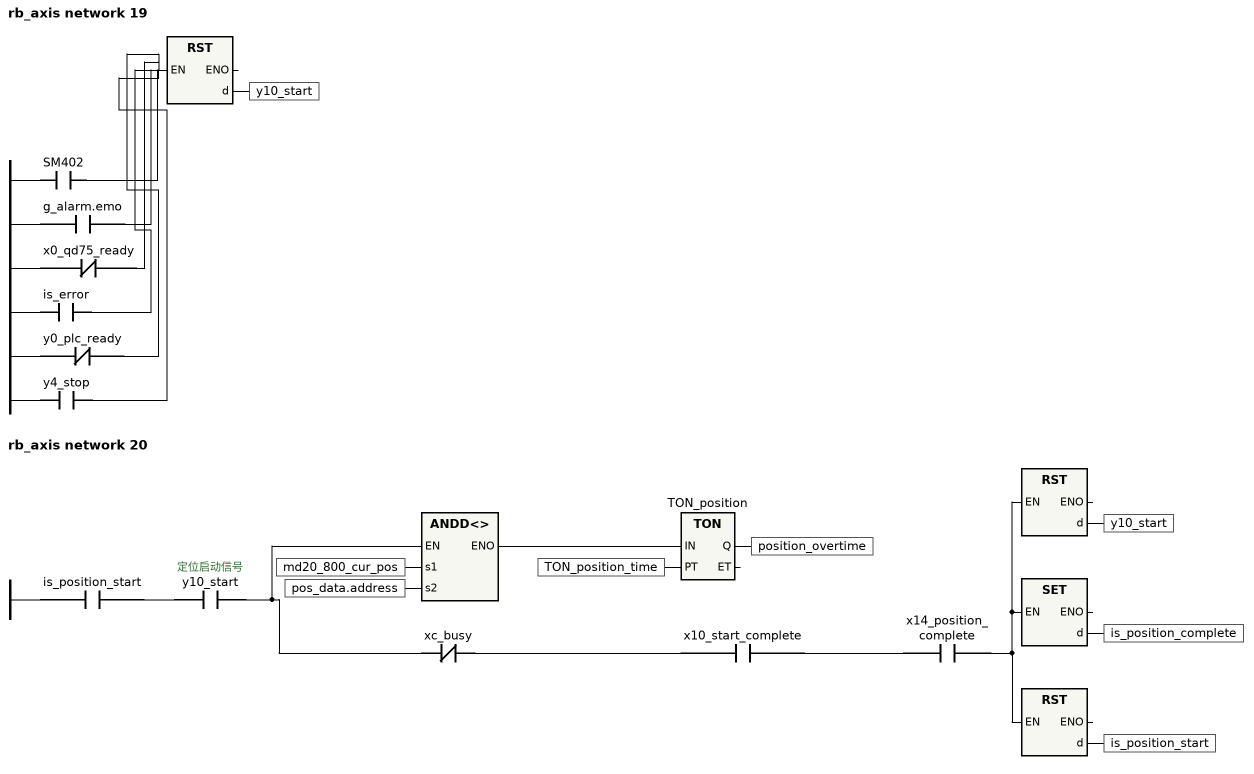
(* network 19 *)
RST(SM402 OR g_alarm.emo OR (NOT x0_qd75_ready) OR is_error OR (NOT y0_plc_ready) OR y4_stop, y10_start);
(* network 20 *)
_p1 := is_position_start AND y10_start;
_p2 := _p1 AND NOT xc_busy AND x10_start_complete AND x14_position_complete;
RST(_p2, y10_start);
SET(_p2, is_position_complete);
_e3 := ANDD<>(_p1, md20_800_cur_pos, pos_data.address);
TON_position(IN := _e3, PT := TON_position_time, Q => position_overtime);
RST(_p2, is_position_start);
END_FUNCTION_BLOCK

FUNCTION calc_address
VAR_INPUT
  index : INT;
  base : INT;
  offset : INT;
END_VAR
calc_address := base + index*offset;
END_FUNCTION

FUNCTION_BLOCK rb_dispatch
VAR
  state : INT;
END_VAR
VAR_INPUT
  first_tid : INT;
  last_tid : INT;
END_VAR
VAR
  tid : INT;
  id1 : INT;
END_VAR
VAR_OUTPUT
  cmd_h_home : BOOL;
  cmd_h_position : BOOL;
  h_address : DINT;
  h_speed : DINT;
  cmd_v_position : BOOL;
  v_address : DINT;
  v_speed : DINT;
END_VAR
VAR_INPUT
  h_is_error : BOOL;
  h_action_enable : BOOL;
  h_position_enable : BOOL;
  h_home_complete : BOOL;
  h_position_complete : BOOL;
  h_cur_pos : DINT;
  v_is_error : BOOL;
  v_action_enable : BOOL;
  v_position_enable : BOOL;
  v_home_complete : BOOL;
  v_position_complete : BOOL;
  v_cur_pos : DINT;
  x_car_sensor1 : BOOL;
  x_car_sensor2 : BOOL;
  x_car_sensor3 : BOOL;
  x_car_sensor4 : BOOL;
END_VAR
VAR
  TON_car_on : TON;
  TON_car_off : TON;
  id2 : INT;
  from_tid : INT;
  to_tid : INT;
  id3 : INT;
  h_address1 : DINT;
  h_address2 : DINT;
END_VAR
VAR_INPUT
  rid : INT;
END_VAR
VAR
  TON_h_home : TON;
  TON_v_home : TON;
  TON_h_position : TON;
  TON_v_position : TON;
  TON_cover : TON;
  TON_car : TON;
  cur_tid : INT;
  TON_rb_inter_lock : TON;
  wait_rb_inter_lock : BOOL;
END_VAR
VAR_OUTPUT
  cmd_h_jog_forward : BOOL;
  cmd_h_jog_reverse : BOOL;
  cmd_v_jog_forward : BOOL;
  cmd_v_jog_reverse : BOOL;
END_VAR
VAR_INPUT
  x_tech_h_forward : BOOL;
  x_tech_h_reverse : BOOL;
  x_tech_v_forward : BOOL;
  x_tech_v_reverse : BOOL;
END_VAR
VAR CONSTANT
  key_h_jog_forward : INT := 10;
  key_h_jog_reverse : INT := 11;
  key_h_jog_high_speed : INT := 12;
  key_h_jog_low_speed : INT := 13;
  key_v_jog_forward : INT := 14;
  key_v_jog_reverse : INT := 15;
  key_v_jog_high_speed : INT := 16;
  key_v_jog_low_speed : INT := 17;
  key_jog_stop : INT := 18;
  key_home : INT := 20;
  key_goto_lock : INT := 21;
  key_goto_unlock : INT := 22;
  key_take : INT := 23;
  key_put : INT := 24;
  key_clean : INT := 25;
  key_teach_enable : INT := 30;
  key_teach_disable : INT := 31;
END_VAR
VAR
  run_list : ARRAY [0..19] OF INT;
END_VAR
VAR_OUTPUT
  cmd_v_home : BOOL;
END_VAR
VAR CONSTANT
  key_add_car : INT := 32;
  key_remove_car : INT := 33;
  key_chuck_on : INT := 34;
  key_chuck_off : INT := 35;
END_VAR
VAR
  is_alarm_take : BOOL;
  is_alarm_put : BOOL;
  is_open_cover_overtime : BOOL;
  is_check_car_overtime : BOOL;
  is_wait_interlock_overtime : BOOL;
  is_tech_box_enable : BOOL;
  is_h_high_speed : BOOL;
  is_v_high_speed : BOOL;
END_VAR
IF SM402 THEN
	cur_tid:=-1;
END_IF;

TON_car_on(IN:=x_car_sensor1 AND x_car_sensor2 AND  x_car_sensor3 AND  x_car_sensor4,PT:=T#1s);
TON_car_off(IN:=NOT x_car_sensor1 AND NOT x_car_sensor2 AND NOT x_car_sensor3 AND NOT x_car_sensor4,PT:=T#1s);
TON_car(IN:=NOT TON_car_on.Q AND NOT TON_car_off.Q,PT:=T#60s);
is_check_car_overtime:=Ton_car.Q;

TON_h_home(IN:=cmd_h_home,PT:=T#300s);
TON_v_home(IN:=cmd_v_home ,PT:=T#180s);

TON_h_position(IN:=cmd_h_position,PT:=T#300s);
TON_v_position(IN:=cmd_v_position,PT:=T#180s);

TON_rb_inter_lock(IN:=wait_rb_inter_lock,PT:=T#180s);
is_wait_interlock_overtime:=TON_rb_inter_lock.Q;

IF g_alarm.emo OR h_is_error OR v_is_error THEN
	FOR  id2 := first_tid TO last_tid BY 1 DO
		IF g_tk_status[id2].rb_inter_lock = rid+1 THEN
			g_tk_status[id2].rb_inter_lock:=0;
		END_IF;
	END_FOR;
	
	run_list[0] := 0;
	
	state:=0;
END_IF;

IF g_sys_status.mmode THEN
	IF g_rb_status[rid].pc_key = key_h_jog_high_speed THEN 
		is_h_high_speed:=TRUE;
	ELSIF g_rb_status[rid].pc_key = key_h_jog_low_speed THEN
		is_h_high_speed:=FALSE;
	ELSIF g_rb_status[rid].pc_key = key_v_jog_high_speed THEN 
		is_v_high_speed:=TRUE;
	ELSIF g_rb_status[rid].pc_key = key_v_jog_low_speed THEN
		is_v_high_speed:=FALSE;
	ELSIF g_rb_status[rid].pc_key = key_teach_enable THEN
		is_tech_box_enable:=TRUE;
	ELSIF g_rb_status[rid].pc_key = key_teach_disable THEN
		is_tech_box_enable:=FALSE;
	ELSIF g_rb_status[rid].pc_key = key_add_car THEN
		g_rb_car[rid].cid:=1;
	ELSIF g_rb_status[rid].pc_key = key_remove_car THEN
		g_rb_car[rid].cid:=0;
	END_IF;
END_IF;

CASE state OF
0:
(**************Idle**************)
cmd_h_jog_forward:= FALSE;
cmd_h_jog_reverse:=FALSE;
cmd_h_home:=FALSE;
cmd_h_position:=FALSE;

cmd_v_jog_forward:= FALSE;
cmd_v_jog_reverse:=FALSE;
cmd_v_home:=FALSE;
cmd_v_position:=FALSE;

IF NOT h_action_enable  OR NOT v_action_enable THEN
	cur_tid:=-1;
	state:=0;
		
ELSIF g_sys_status.mmode AND g_rb_status[rid].pc_key = key_h_jog_forward THEN
		state:= 10;	
ELSIF g_sys_status.mmode AND is_tech_box_enable AND x_tech_h_forward THEN
		state:= 11;		
ELSIF g_sys_status.mmode AND g_rb_status[rid].pc_key = key_h_jog_reverse THEN
		state:= 12;
ELSIF g_sys_status.mmode AND is_tech_box_enable AND x_tech_h_reverse THEN
		state:= 13;
ELSIF g_sys_status.mmode AND g_rb_status[rid].pc_key = key_v_jog_forward THEN
		state:= 14;	
ELSIF g_sys_status.mmode AND is_tech_box_enable AND x_tech_v_forward THEN
		state:= 15;			
ELSIF g_sys_status.mmode AND g_rb_status[rid].pc_key = key_v_jog_reverse THEN
		state:= 16;		
ELSIF g_sys_status.mmode AND is_tech_box_enable AND x_tech_v_reverse THEN
		state:= 17;		
ELSIF g_sys_status.mmode AND  g_rb_status[rid].pc_key = key_home THEN 
		state:= 100;
			
ELSIF NOT h_position_enable OR NOT v_position_enable THEN
	cur_tid:=-1;
	IF g_sys_status.amode AND g_sys_status.enable_run THEN
		state:= 100;
	END_IF;
		
ELSIF g_sys_status.amode AND g_sys_status.enable_run THEN
	IF run_list[0] > 0 THEN
		FIFR(TRUE,state, run_list[0]);
		FIFR(TRUE,tid, run_list[0]);
	ELSE 
		state := 1000;
	END_IF;
	
ELSIF g_sys_status.mmode THEN
	IF g_rb_status[rid].pc_key=key_goto_lock THEN
		tid:=g_rb_status[rid].pc_tid;
		state :=  200;
	
	ELSIF g_rb_status[rid].pc_key=key_goto_unlock THEN
		tid:=g_rb_status[rid].pc_tid;
		state :=  300;
	
	ELSIF g_rb_status[rid].pc_key=key_take THEN
		tid:=g_rb_status[rid].pc_tid;
		state :=  400;
	
	ELSIF g_rb_status[rid].pc_key=key_put THEN
		tid:=g_rb_status[rid].pc_tid;
		state :=  500;
	
	ELSIF g_rb_status[rid].pc_key=key_clean THEN
		state :=  600;
	END_IF;
	
END_IF;	

10:
cmd_h_jog_forward := TRUE;
IF g_rb_status[rid].pc_key = key_jog_stop  THEN
	cmd_h_jog_forward :=FALSE;
	state :=  0;
END_IF;
11:
IF x_tech_h_forward THEN
	cmd_h_jog_forward :=TRUE;
ELSE
	cmd_h_jog_forward :=FALSE;
	state :=  0;		
END_IF;
12:
cmd_h_jog_reverse := TRUE;
IF g_rb_status[rid].pc_key = key_jog_stop THEN
	cmd_h_jog_reverse :=FALSE;
	state :=  0;
END_IF;
13:
cmd_h_jog_reverse := TRUE;
IF NOT x_tech_h_reverse THEN
	cmd_h_jog_reverse :=FALSE;
	state :=  0;
END_IF;
14:
cmd_v_jog_forward := TRUE;
IF g_rb_status[rid].pc_key = key_jog_stop THEN
	cmd_v_jog_forward :=FALSE;
	state :=  0;
END_IF;
15:
cmd_v_jog_forward := TRUE;
IF NOT x_tech_v_forward THEN
	cmd_v_jog_forward :=FALSE;
	state :=  0;
END_IF;
16:
cmd_v_jog_reverse := TRUE;
IF g_rb_status[rid].pc_key = key_jog_stop THEN
	cmd_v_jog_reverse :=FALSE;
	state :=  0;
END_IF;
17:
cmd_v_jog_reverse := TRUE;
IF NOT x_tech_v_reverse THEN
	cmd_v_jog_reverse :=FALSE;
	state :=  0;
END_IF;

100:
(*************Home State*************)
cmd_v_home:=TRUE;
state :=  101;

101:
IF v_home_complete AND v_cur_pos = 0 THEN
	cmd_v_home:=FALSE;
	cmd_h_home:=TRUE;
	state :=  102;
END_IF;

102:
IF h_home_complete AND h_cur_pos = 0 THEN
	cmd_h_home:=FALSE;
	state :=  0;
END_IF;

200:
(************Goto Lock State************)
IF first_tid > 0 AND tid = first_tid THEN 
	h_address1 :=  g_tk_pos[tid].h_lock2;
ELSE
	h_address1 :=  g_tk_pos[tid].h_lock;
END_IF;
state:= 201;

201:
IF v_cur_pos = g_safe_height THEN
	state:= 203;
ELSE
	v_address := g_safe_height;
	v_speed := rb_speed(FALSE,FALSE, g_rb_car[rid].cid,tid);
	cmd_v_position:=TRUE;
	state:= 202;
END_IF;

202:
IF v_position_complete AND v_cur_pos = g_safe_height THEN
	cmd_v_position:=FALSE;
	state:=203;
END_IF;

203:
IF h_cur_pos = h_address1 THEN
	g_tk_status[tid].rb_inter_lock := rid+1;
	cur_tid:=tid;
	state := 0;
ELSIF g_tk_status[tid].rb_inter_lock=0 OR g_tk_status[tid].rb_inter_lock = rid+1THEN 
	wait_rb_inter_lock:=FALSE;
	g_tk_status[tid].rb_inter_lock := rid+1;
	h_address := h_address1;
	h_speed := rb_speed(TRUE,TRUE,g_rb_car[rid].cid,tid);
	cmd_h_position:=TRUE;
	state:= 204;
ELSE
	wait_rb_inter_lock:=TRUE;
END_IF;

204:
IF h_cur_pos = h_address1 AND h_position_complete THEN
	IF cur_tid <>-1 THEN
		g_tk_status[cur_tid].rb_inter_lock := 0;
	END_IF;
	
	cur_tid:=tid;
	g_tk_status[tid].rb_inter_lock := rid+1;
	
	cmd_h_position:=FALSE;
	state := 0;
END_IF;


300:
(*************Goto Unlock State*************)
IF first_tid > 0 AND tid = first_tid THEN 
	h_address1 :=  g_tk_pos[tid].h_unlock2;
ELSE
	h_address1 :=  g_tk_pos[tid].h_unlock;
END_IF;

state:= 201;

400:
(*************Take State*************)
IF first_tid > 0 AND tid = first_tid THEN 
	h_address1 :=  g_tk_pos[tid].h_unlock2;
	h_address2 :=  g_tk_pos[tid].h_lock2;
ELSE
	h_address1 :=  g_tk_pos[tid].h_unlock;
	h_address2 :=  g_tk_pos[tid].h_lock;
END_IF;

IF g_rb_car[rid].cid = 0 THEN 
	state :=  401;
ELSE
	is_alarm_take:= TRUE;
	IF g_sys_status.key_reset AND g_sys_status.mmode THEN
		is_alarm_take:= FALSE;
		run_list[0] := 0;
		state := 0;	
	END_IF;
END_IF;

401:
IF v_cur_pos = g_safe_height THEN
	state:= 403;
ELSE
	v_address := g_safe_height;
	v_speed := rb_speed(FALSE,FALSE,g_rb_car[rid].cid,tid);
	cmd_v_position:=TRUE;
	state:= 402;
END_IF;

402:
IF v_position_complete AND v_cur_pos = g_safe_height THEN
	cmd_v_position:=FALSE;
	state:=403;
END_IF;

403:
IF h_cur_pos = h_address1 THEN
	g_tk_status[tid].cmd_open_cover:=TRUE;
	g_tk_status[tid].cmd_close_cover:=FALSE;
	g_tk_status[tid].rb_inter_lock := rid+1;
	cur_tid:=tid;
	state :=405;
ELSIF g_tk_status[tid].rb_inter_lock=0 OR g_tk_status[tid].rb_inter_lock = rid+1THEN 
	g_tk_status[tid].cmd_open_cover:=TRUE;
	g_tk_status[tid].cmd_close_cover:=FALSE;
	wait_rb_inter_lock:=FALSE;
	g_tk_status[tid].rb_inter_lock := rid+1;
	
	h_address := h_address1;
	h_speed := rb_speed(TRUE,TRUE,g_rb_car[rid].cid,tid);
	cmd_h_position:=TRUE;
	state:= 404;
ELSE 
	wait_rb_inter_lock:=TRUE;
END_IF;

404:
IF h_cur_pos = h_address1 AND h_position_complete THEN
	IF cur_tid <>-1 THEN
		g_tk_status[cur_tid].rb_inter_lock := 0;
	END_IF;
	
	cur_tid:=tid;
	g_tk_status[tid].rb_inter_lock := rid+1;
	
	cmd_h_position:=FALSE;
	state := 405;
END_IF;

405:
TON_cover(IN:=g_tk_status[tid].cmd_open_cover AND NOT g_tk_status[tid].cover_is_open,PT:=T#120s);
is_open_cover_overtime:=TON_cover.Q;
IF g_tk_status[tid].cover_is_open THEN
	state:=406;
ELSIF TON_cover.Q AND  g_sys_status.key_reset AND g_sys_status.mmode THEN
	g_tk_status[tid].cmd_open_cover:=FALSE;
	g_tk_status[tid].cmd_close_cover:=FALSE;
	run_list[0] := 0;
	state := 0;	
END_IF;
	
406:
IF first_tid > 0 AND tid = first_tid THEN 
	v_address := g_tk_pos[tid].v_bottom2;
ELSE
	v_address := g_tk_pos[tid].v_bottom;
END_IF;

v_speed := rb_speed(FALSE,FALSE,g_rb_car[rid].cid,tid);
cmd_v_position:=TRUE;
state:= 407;
	
407:
IF v_position_complete AND v_cur_pos = v_address THEN
	cmd_v_position:=FALSE;
	state:=408;
END_IF;

408:
	h_address := h_address2;
	h_speed := rb_speed(TRUE,FALSE,g_rb_car[rid].cid,tid);
	cmd_h_position:=TRUE;
	state:= 409;
	
409:
IF h_cur_pos = h_address2 AND h_position_complete THEN
	cmd_h_position:=FALSE;
	state := 410;
END_IF;

410:
IF TON_car_on.Q  AND (h_address2 =  g_tk_pos[tid].h_lock OR h_address2 =  g_tk_pos[tid].h_lock2 ) THEN
	(*take flow*)
	g_tk_car[tid].leave_time[tid]:=2;
	g_rb_car[rid] := g_tk_car[tid];
	g_tk_car[tid].cid := 0;
	state := 411;

ELSIF TON_car_off.Q  AND (h_address2 =  g_tk_pos[tid].h_unlock OR h_address2 =  g_tk_pos[tid].h_unlock2) THEN
	(*put flow*)
	g_tk_car[tid] := g_rb_car[rid];
	g_tk_car[tid].enter_time[tid]:=1;
	g_rb_car[rid].cid := 0;
	state := 411;

ELSIF TON_car.Q  AND g_sys_status.key_reset AND g_sys_status.mmode THEN
	run_list[0] := 0;
	state := 411;	
END_IF;


411:
	v_address := g_safe_height;
	v_speed := rb_speed(FALSE,FALSE,g_rb_car[rid].cid,tid);
	cmd_v_position:=TRUE;
	state:= 412;

412:
IF v_position_complete AND v_cur_pos = g_safe_height THEN
	cmd_v_position:=FALSE;
	g_tk_status[tid].cmd_open_cover:=FALSE;
	g_tk_status[tid].cmd_close_cover:=TRUE;
	state:=0;

(*	
	IF first_tid > 0 AND tid = first_tid THEN 
		tid:=tid+1;
		h_address1 :=  g_tk_pos[tid].h_unlock;
		state:=413;
	ELSIF tid = last_tid THEN 
		tid:=tid-1;
		h_address1 :=  g_tk_pos[tid].h_unlock;
		state:=413;
	ELSE
		state:=0;
	END_IF;
*)	
END_IF;

413:
IF g_tk_status[tid].rb_inter_lock=0 OR g_tk_status[tid].rb_inter_lock = rid+1THEN 
	wait_rb_inter_lock:=FALSE;
	g_tk_status[tid].rb_inter_lock := rid+1;
	h_address := h_address1;
	h_speed := rb_speed(TRUE,TRUE,g_rb_car[rid].cid,tid);
	cmd_h_position:=TRUE;
	state:= 414;
ELSE 
	wait_rb_inter_lock:=TRUE;
END_IF;

IF TON_rb_inter_lock.Q AND g_sys_status.key_reset AND g_sys_status.mmode THEN 
	wait_rb_inter_lock:=FALSE;
	run_list[0] := 0;
	state:=0;
END_IF;

414:
IF h_cur_pos = h_address1 AND h_position_complete THEN
	IF cur_tid <>-1 THEN
		g_tk_status[cur_tid].rb_inter_lock := 0;
	END_IF;
	
	cur_tid:=tid;
	g_tk_status[tid].rb_inter_lock := rid+1;
	
	cmd_h_position:=FALSE;
	state := 0;
END_IF;

500:
(*************Put State*************)
IF first_tid > 0 AND tid = first_tid THEN 
	h_address1 :=  g_tk_pos[tid].h_lock2;
	h_address2 :=  g_tk_pos[tid].h_unlock2;
ELSE
	h_address1 :=  g_tk_pos[tid].h_lock;
	h_address2 :=  g_tk_pos[tid].h_unlock;
END_IF;

IF g_rb_car[rid].cid <> 0 THEN 
	state :=  401;
ELSE
	is_alarm_put:= TRUE;
	IF g_sys_status.key_reset AND g_sys_status.mmode THEN
		is_alarm_put:= FALSE;
		run_list[0] := 0;
		state := 0;	
	END_IF;
END_IF;

600:
(*************Clean State*************)
state :=  0;


1000:
(*************Search State*************)
from_tid := -1;
to_tid := -1;

FOR  id1 := first_tid TO last_tid-1 BY 1 DO
	IF (from_tid=-1 
		OR g_tk_cnf[id1].take_weight > g_tk_cnf[from_tid].take_weight 
		OR ( g_tk_cnf[id1].take_weight = g_tk_cnf[from_tid].take_weight AND g_tk_car[id1].proc_time[id1] < g_tk_car[from_tid].proc_time[from_tid] )) 
		AND g_tk_car[id1].cid>0  AND g_tk_car[id1].proc_time[id1] <= 0 
		AND g_tk_status[id1].permit_take AND g_tk_status[id1].rb_inter_lock=0 THEN
		
		FOR  id2 := 0 TO 4 BY 1 DO
			id3 :=  g_tk_cnf[id1].next_tank[id2];
			IF id3>id1 AND g_tk_car[id3].cid=0  AND g_tk_status[id3].permit_put AND g_tk_status[id3].rb_inter_lock=0 THEN
				from_tid := id1;
				to_tid := id3;
				EXIT;
			END_IF;
		END_FOR;
		
	END_IF;
END_FOR;

IF from_tid >= first_tid  AND from_tid<last_tid 
	AND to_tid>first_tid AND to_tid <= last_tid THEN
	
	FIFW(TRUE,400, run_list[0]);
	FIFW(TRUE,from_tid, run_list[0]);
	FIFW(TRUE,500, run_list[0]);
	FIFW(TRUE,to_tid, run_list[0]);
	
	IF to_tid = last_tid THEN
		FIFW(TRUE,300, run_list[0]);
		FIFW(TRUE,to_tid-1, run_list[0]);
	END_IF;
END_IF;

state :=  0;

END_CASE;

g_rb_status[rid].pc_key:=0;
END_FUNCTION_BLOCK

FUNCTION rb_speed
VAR_INPUT
  tid : INT;
END_VAR
VAR CONSTANT
  h_high_speed : DINT;
  h_mid_speed : DINT;
  h_low_speed : DINT;
  v_high_speed : DINT;
  v_mid_speed : DINT;
  v_low_speed : DINT;
END_VAR
VAR_INPUT
  is_axis_h : BOOL;
  is_safe_height : BOOL;
  car_id : INT;
END_VAR
IF is_axis_h  THEN
	IF is_safe_height THEN
			IF car_id >0 THEN
				rb_speed :=  h_mid_speed;
			ELSE
				rb_speed := h_high_speed;
			END_IF;
	ELSE
			IF car_id>0 THEN
				rb_speed :=  h_low_speed;
			ELSE
				rb_speed :=h_low_speed;
			END_IF;
	END_IF;
ELSE
	IF is_safe_height THEN
			IF car_id>0 THEN
				rb_speed :=  v_low_speed;
			ELSE
				rb_speed := v_high_speed;
			END_IF;
	ELSE
			IF car_id>0 THEN
				rb_speed :=  v_low_speed;
			ELSE
				rb_speed :=v_high_speed;
			END_IF;
	END_IF;
END_IF;
END_FUNCTION

FUNCTION_BLOCK fb_cover
VAR_INPUT
  bAuto : BOOL;
  bACmd : BOOL;
  S_L_Op : BOOL;
  S_L_Cl : BOOL;
  S_R_Op : BOOL;
  S_R_Cl : BOOL;
  Interlock : BOOL;
  KeyOpen : BOOL;
  KeyReset : BOOL;
  MoveTimeout : TIME;
END_VAR
VAR_OUTPUT
  Valve_L_Op : BOOL;
  Valve_L_Cl : BOOL;
  F_SensorError : BOOL;
  F_Timeout : BOOL;
  W_SensorError : BOOL;
  ReadyOp : BOOL;
  ReadyCl : BOOL;
END_VAR
VAR
  state : INT;
  TON_Switch : TON;
  Fault_Timeout : TON;
  Fault_Sensor : TON;
  TON_Ready_Op : TON;
  TON_Ready_Cl : TON;
  TON_Open : TON;
  TON_Close : TON;
END_VAR

TON_Open(IN:=S_L_Op AND S_R_Op AND NOT S_L_Cl AND  NOT S_L_Cl  ,PT:=T#500ms);
TON_Close(IN:=NOT S_L_Op AND NOT S_R_Op AND  S_L_Cl AND   S_L_Cl  ,PT:=T#500ms);

Fault_Timeout ( IN:=  (Valve_L_Op AND NOT  S_L_Op) OR
					 (Valve_L_Op AND NOT  S_R_Op) OR
					 (Valve_L_Cl AND NOT  S_L_Cl) OR
					 (Valve_L_Cl AND NOT  S_R_Cl)  AND NOT KeyReset ,
				PT := MoveTimeout);


F_Timeout :=Fault_Timeout.Q;

Fault_Sensor( IN:= (S_L_Op AND S_L_Cl) OR  (S_R_Op AND S_R_Cl)   AND NOT KeyReset,
			PT := MoveTimeout);


IF F_Timeout THEN
state := 0;
END_IF;


IF KeyReset THEN
	W_SensorError := FALSE;
END_IF;


CASE state OF
0:
	Valve_L_Op  := FALSE;
	Valve_L_Cl :=FALSE;

	IF S_L_Op AND S_R_Op AND NOT S_L_Cl AND  NOT S_R_Cl THEN
		state := 10;
		W_SensorError := FALSE;
	ELSIF NOT S_L_Op AND NOT S_R_Op AND  S_L_Cl AND   S_R_Cl THEN
		state := 20;
		W_SensorError := FALSE;
	ELSE
		W_SensorError := TRUE;
	END_IF;
	
	IF KeyOpen AND Interlock  AND NOT bAuto THEN
		IF 	Valve_L_Op  THEN
			Valve_L_Op := FALSE;
			Valve_L_Cl :=TRUE;
		ELSE
				Valve_L_Op  := TRUE;
				Valve_L_Cl :=FALSE;
		END_IF;
	END_IF;


(*Cover Open State*)
10:
	Valve_L_Op  := TRUE;
	Valve_L_Cl :=FALSE;
	IF KeyOpen AND Interlock  AND NOT bAuto THEN
		state := 11;
	ELSIF bAuto AND NOT bACmd THEN
		state := 11;
	END_IF;
(* Open -> Close *)
11:
	Valve_L_Op  := FALSE;
	Valve_L_Cl :=TRUE;
	IF KeyOpen AND NOT bAuto  THEN
		state := 10;
	ELSIF TON_Close.Q THEN
		state := 20;
	END_IF;
(*Clsoe State*)
20:
	Valve_L_Op  := FALSE;
	Valve_L_Cl :=TRUE;
	IF KeyOpen AND  Interlock  AND NOT bAuto  THEN
		state := 21;
	ELSIF bAuto AND  bACmd THEN
		state := 21;
	END_IF;

21:
	Valve_L_Op  := TRUE;
	Valve_L_Cl :=FALSE;
	IF NOT KeyOpen AND NOT bAuto  THEN
		state := 20;
	ELSIF TON_Open.Q THEN
		state := 10;
	END_IF;

END_CASE;


TON_Ready_Op(IN :=  S_L_Op AND S_R_Op AND NOT S_L_Cl AND NOT S_R_Cl AND NOT Valve_L_Cl ,
				PT := T#200ms);

ReadyOp := TON_Ready_Op.Q;
TON_Ready_Cl(IN:= NOT S_L_Op AND NOT  S_R_Op AND  S_L_Cl AND S_R_Cl AND NOT Valve_L_Op,
				PT := T#200ms);

ReadyCl := TON_Ready_Cl.Q;
END_FUNCTION_BLOCK

FUNCTION_BLOCK pc_comm
VAR
  rid : INT;
  tid : INT;
END_VAR
VAR CONSTANT
  key_save_h_lock : INT := 40;
  key_save_h_unlock : INT := 41;
  key_save_v_bottom : INT := 42;
  key_save_h_lock2 : INT := 43;
  key_save_h_unlock2 : INT := 44;
  key_save_v_bottom2 : INT := 45;
  key_save_pc_h_lock : INT := 50;
  key_save_pc_h_unlock : INT := 51;
  key_save_pc_v_bottom : INT := 52;
  key_save_pc_h_lock2 : INT := 53;
  key_save_pc_h_unlock2 : INT := 54;
  key_save_pc_v_bottom2 : INT := 55;
END_VAR
VAR
  pc_key : INT;
  pc_tank_pos : DINT;
END_VAR
CASE g_pc_cmd[0] OF
	
(*robot command*)	
10:
rid:= g_pc_cmd[1];
g_rb_status[rid].pc_key := g_pc_cmd[2];
g_rb_status[rid].pc_tid := g_pc_cmd[3];

g_pc_cmd[0]:=18;

(*save robot pos from qd75*)
40:
rid:= g_pc_cmd[1];
tid:= g_pc_cmd[2];
pc_key := g_pc_cmd[3];

IF pc_key = key_save_h_lock THEN(*x lock position*)
	g_tk_pos[tid].h_lock:= g_rb_status[rid].h_cur_pos;
END_IF;

IF pc_key = key_save_h_unlock THEN(*x  unlock position*)
	g_tk_pos[tid].h_unlock:= g_rb_status[rid].h_cur_pos;
END_IF;

IF pc_key = key_save_v_bottom THEN(*z  bottom position*)
	g_tk_pos[tid].v_bottom:= g_rb_status[rid].v_cur_pos;
END_IF;

IF pc_key = key_save_h_lock2 THEN(*x lock position2*)
	g_tk_pos[tid].h_lock2:= g_rb_status[rid].h_cur_pos;
END_IF;

IF pc_key = key_save_h_unlock2 THEN(*x  unlock position2*)
	g_tk_pos[tid].h_unlock2:= g_rb_status[rid].h_cur_pos;
END_IF;

IF pc_key = key_save_v_bottom2 THEN(*z  bottom position2*)
	g_tk_pos[tid].v_bottom2:= g_rb_status[rid].v_cur_pos;
END_IF;

g_pc_cmd[0]:=48;


(*save robot pos from pc *)
50:
rid:= g_pc_cmd[1];
tid:= g_pc_cmd[2];
pc_key := g_pc_cmd[3];

D0:=g_pc_cmd[4];
D1:=g_pc_cmd[5];
DMOV(TRUE,D0,pc_tank_pos);

IF pc_key = key_save_pc_h_lock THEN(*x lock position*)
	g_tk_pos[tid].h_lock:=pc_tank_pos;
END_IF;

IF pc_key= key_save_pc_h_unlock THEN(*x  unlock position*)
	g_tk_pos[tid].h_unlock:=pc_tank_pos;
END_IF;

IF pc_key = key_save_pc_v_bottom THEN(*z  bottom position*)
	g_tk_pos[tid].v_bottom:=pc_tank_pos;
END_IF;

IF pc_key = key_save_pc_h_lock2 THEN(*x lock position2*)
	g_tk_pos[tid].h_lock2:=pc_tank_pos;
END_IF;

IF pc_key = key_save_pc_h_unlock2 THEN(*x  unlock position2*)
	g_tk_pos[tid].h_unlock2:=pc_tank_pos;
END_IF;

IF pc_key = key_save_pc_v_bottom2 THEN(*z  bottom position2*)
	g_tk_pos[tid].v_bottom2:=pc_tank_pos;
END_IF;

g_pc_cmd[0]:=58;


(*tank manual op*)
200:
tid:= g_pc_cmd[1];

g_pc_cmd[0]:=208;


END_CASE;
END_FUNCTION_BLOCK

FUNCTION_BLOCK tk_diw
VAR_INPUT
  tid : INT;
END_VAR
VAR_OUTPUT
  y_fill_up : BOOL;
  y_fill_down : BOOL;
  y_bubble : BOOL;
  y_drain : BOOL;
END_VAR
VAR_INPUT
  x_level_high : BOOL;
  x_level_low : BOOL;
  x_water_alarm : BOOL;
END_VAR
VAR
  valve_fill_up : fb_valve;
  valve_fill_down : fb_valve;
  valve_bubble : fb_valve;
  valve_drain : fb_valve;
  fb_qdr_1 : fb_qdr;
  interlock : BOOL;
END_VAR
VAR CONSTANT
  key_qdr : INT;
  key_fill_up : INT;
  key_fill_down : INT;
  key_bubble : INT;
  key_drain : INT;
END_VAR
VAR
  fb_cover_1 : fb_cover;
END_VAR
(* structured ladder/FBD written out as ST: instructions are called as NAME(EN, inputs, outputs); _pN, _eN, _tN stand for wires *)
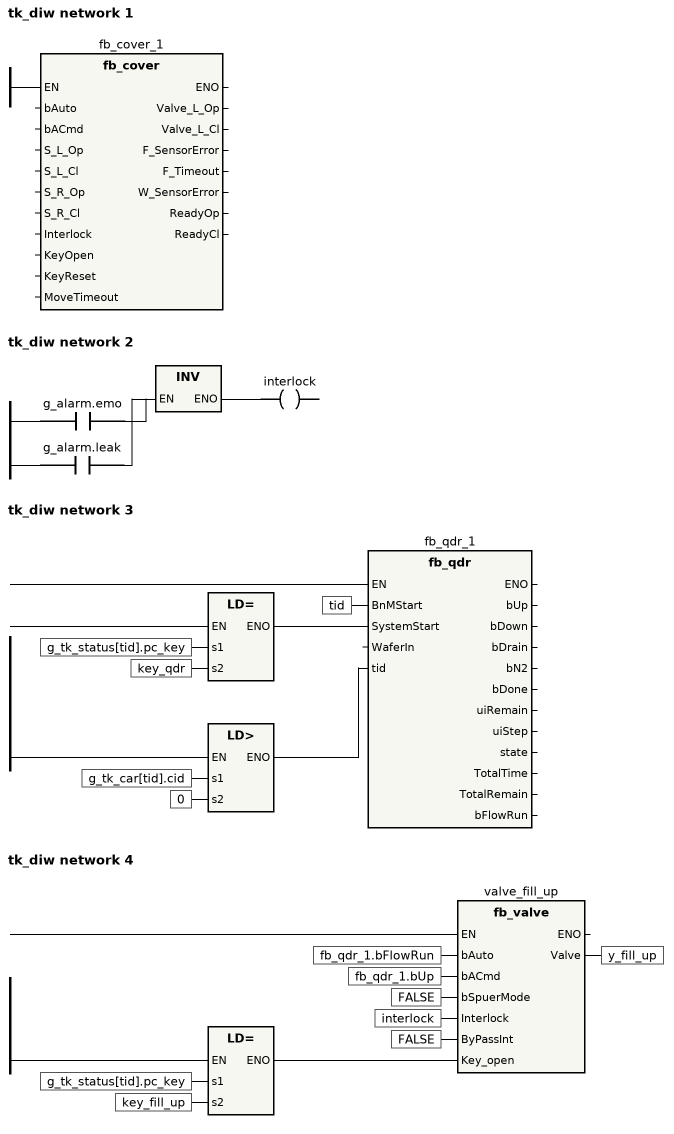
(* network 1 *)
fb_cover_1(EN := TRUE);
(* network 2 *)
_e1 := INV(g_alarm.emo OR g_alarm.leak);
interlock := _e1;
(* network 3 *)
_e1 := LD=(TRUE, g_tk_status[tid].pc_key, key_qdr);
_e2 := LD>(TRUE, g_tk_car[tid].cid, 0);
fb_qdr_1(EN := TRUE, BnMStart := tid, SystemStart := _e1, tid := _e2);
(* network 4 *)
_e1 := LD=(TRUE, g_tk_status[tid].pc_key, key_fill_up);
valve_fill_up(EN := TRUE, bAuto := fb_qdr_1.bFlowRun, bACmd := fb_qdr_1.bUp, bSpuerMode := FALSE, Interlock := interlock, ByPassInt := FALSE, Key_open := _e1, Valve => y_fill_up);
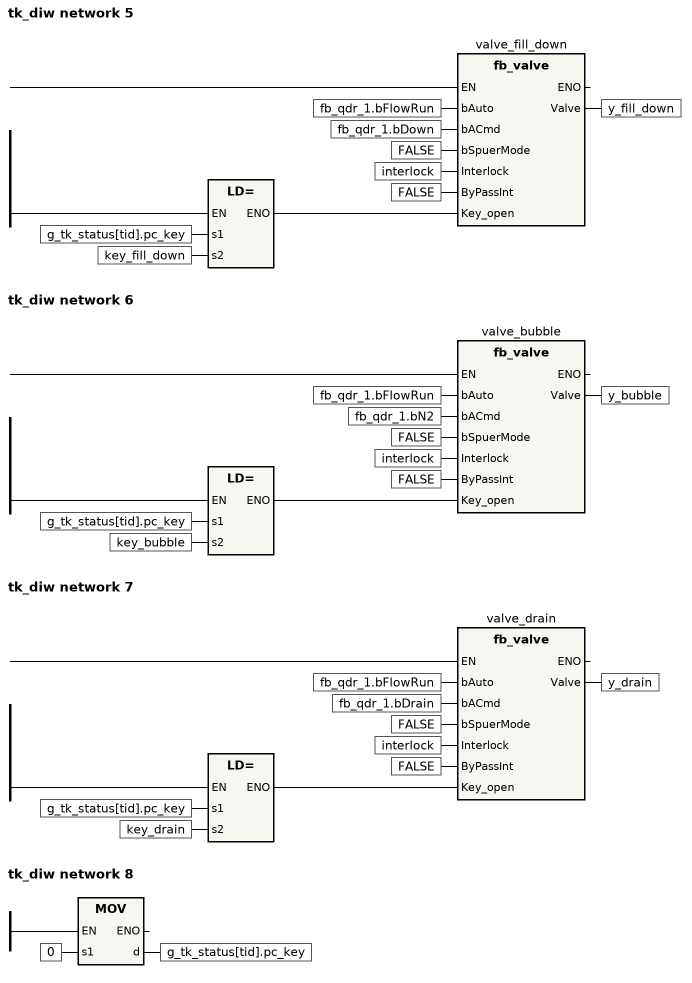
(* network 5 *)
_e1 := LD=(TRUE, g_tk_status[tid].pc_key, key_fill_down);
valve_fill_down(EN := TRUE, bAuto := fb_qdr_1.bFlowRun, bACmd := fb_qdr_1.bDown, bSpuerMode := FALSE, Interlock := interlock, ByPassInt := FALSE, Key_open := _e1, Valve => y_fill_down);
(* network 6 *)
_e1 := LD=(TRUE, g_tk_status[tid].pc_key, key_bubble);
valve_bubble(EN := TRUE, bAuto := fb_qdr_1.bFlowRun, bACmd := fb_qdr_1.bN2, bSpuerMode := FALSE, Interlock := interlock, ByPassInt := FALSE, Key_open := _e1, Valve => y_bubble);
(* network 7 *)
_e1 := LD=(TRUE, g_tk_status[tid].pc_key, key_drain);
valve_drain(EN := TRUE, bAuto := fb_qdr_1.bFlowRun, bACmd := fb_qdr_1.bDrain, bSpuerMode := FALSE, Interlock := interlock, ByPassInt := FALSE, Key_open := _e1, Valve => y_drain);
(* network 8 *)
MOV(TRUE, 0, g_tk_status[tid].pc_key);
END_FUNCTION_BLOCK

FUNCTION_BLOCK fb_valve
VAR
  ValveOut : BOOL;
  F_TRIG_AutoOff : F_TRIG;
  R_TRIG_AutoOn : R_TRIG;
  R_TRIG_bACmdOn : R_TRIG;
END_VAR
VAR_OUTPUT
  Valve : BOOL;
END_VAR
VAR_INPUT
  bAuto : BOOL;
  bACmd : BOOL;
  bSpuerMode : BOOL;
  Interlock : BOOL;
  ByPassInt : BOOL;
  Key_open : BOOL;
END_VAR
VAR
  F_TRIG_bACmdOff : F_TRIG;
END_VAR
F_TRIG_AutoOff(_CLK := bAuto);
R_TRIG_AutoOn(_CLK := bAuto);
R_TRIG_bACmdOn(_CLK :=  bACmd);
F_TRIG_bACmdOff( _CLK := bACmd);

IF R_TRIG_AutoOn.Q THEN
	ValveOut :=bACmd;
END_IF;

IF F_TRIG_AutoOff.Q  THEN
	ValveOut := FALSE;
END_IF;

IF R_TRIG_bACmdOn.Q  AND   bAuto THEN
		ValveOut := TRUE;
END_IF;

IF F_TRIG_bACmdOff.Q  AND   bAuto THEN
		ValveOut := FALSE;
END_IF;

IF Key_open THEN
	IF  bAuto THEN
		IF bSpuerMode THEN
			ValveOut := NOT ValveOut;
		END_IF;
	ELSE
		ValveOut := NOT ValveOut;
	END_IF;
END_IF;

IF Interlock OR  ByPassInt THEN
	Valve := ValveOut;
ELSE
	IF NOT bAuto THEN
		ValveOut := FALSE;
	END_IF;
	Valve := FALSE;
END_IF;
END_FUNCTION_BLOCK

FUNCTION_BLOCK fb_fault
VAR_INPUT
  input : BOOL;
  delay_time : TIME;
  ack : BOOL;
END_VAR
VAR_OUTPUT
  fault : BOOL;
END_VAR
VAR
  TON_set : TON;
END_VAR
(* structured ladder/FBD written out as ST: instructions are called as NAME(EN, inputs, outputs); _pN, _eN, _tN stand for wires *)
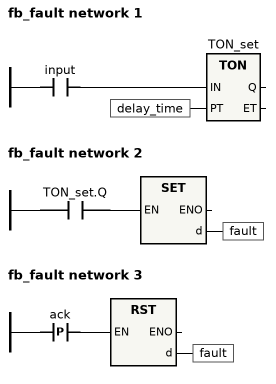
(* network 1 *)
TON_set(IN := input, PT := delay_time);
(* network 2 *)
SET(TON_set.Q, fault);
(* network 3 *)
RST(LDP(TRUE, ack), fault);
END_FUNCTION_BLOCK

PROGRAM main
VAR
  fb_fault_EMG : fb_fault;
  R_TRIG_reset : R_TRIG;
  fb_fault_leak : fb_fault;
  tk_diw_1 : tk_diw;
  pc_comm_1 : pc_comm;
END_VAR
(* structured ladder/FBD written out as ST: instructions are called as NAME(EN, inputs, outputs); _pN, _eN, _tN stand for wires *)
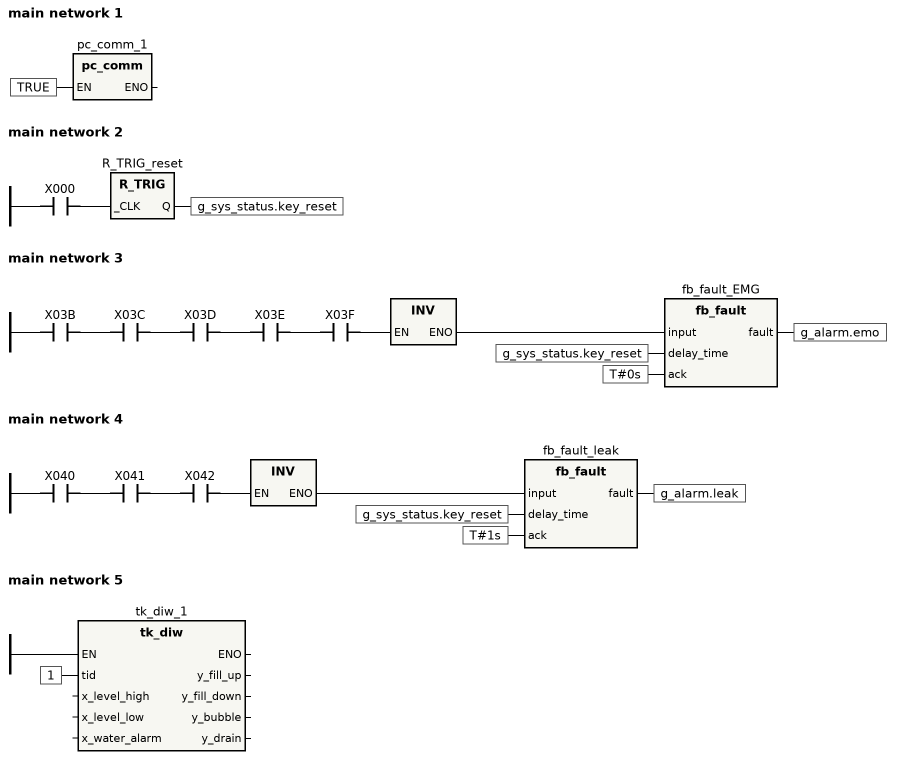
(* network 1 *)
pc_comm_1(EN := TRUE);
(* network 2 *)
R_TRIG_reset(_CLK := X000, Q => g_sys_status.key_reset);
(* network 3 *)
_e1 := INV(X03B AND X03C AND X03D AND X03E AND X03F);
fb_fault_EMG(input := _e1, delay_time := g_sys_status.key_reset, ack := T#0s, fault => g_alarm.emo);
(* network 4 *)
_e1 := INV(X040 AND X041 AND X042);
fb_fault_leak(input := _e1, delay_time := g_sys_status.key_reset, ack := T#1s, fault => g_alarm.leak);
(* network 5 *)
tk_diw_1(EN := TRUE, tid := 1);
END_PROGRAM

FUNCTION_BLOCK fb_qdr
VAR_INPUT
  BnMStart : BOOL;
  SystemStart : BOOL;
  WaferIn : BOOL;
END_VAR
VAR_OUTPUT
  bUp : BOOL;
  bDown : BOOL;
  bDrain : BOOL;
  bN2 : BOOL;
  bDone : BOOL;
  uiRemain : INT;
  uiStep : INT;
  state : INT;
  TotalTime : INT;
  TotalRemain : INT;
END_VAR
VAR
  TotalStepRemain : INT;
  LoopCount : INT;
  R_TRIG_1SEC : R_TRIG;
END_VAR
VAR_OUTPUT
  bFlowRun : BOOL;
END_VAR
VAR
  uiCmd : INT;
END_VAR
VAR_INPUT
  tid : INT;
END_VAR
VAR
  rcp : DIW_RCP;
END_VAR
R_TRIG_1SEC(_CLK :=SM412);

CASE state OF
0:(**)
	bUp := FALSE;
	bDown:=FALSE;
	bDrain := FALSE;
	bN2  := FALSE;
	
	uiStep := 0;
	bDone := FALSE;
	bFlowRun := FALSE;

	IF BnMStart  AND NOT SystemStart THEN
		state:=1;
		uiStep := 0;
		bFlowRun := TRUE;
	ELSIF WaferIn AND SystemStart THEN
		state:=1;
		uiStep := 0;
		bFlowRun := TRUE;
	END_IF;

1:(*Read Recipe*)
		state:=10;
		uiStep :=  uiStep+1;
		BMOV(SM400,g_recipe.tk_data[(tid-1)*g_rcp_max_size],g_rcp_max_size,rcp.LoopCount);
		LoopCount :=rcp.LoopCount;
	 	TotalTime := rcp.uiRemain[0] + 
	 		(rcp.uiRemain[1]+ rcp.uiRemain[2]+rcp.uiRemain[3])*(LoopCount+1) +
	 		rcp.uiRemain[4]+
	 		rcp.uiRemain[5];
		TotalStepRemain := TotalTime;
		TotalRemain :=TotalTime;
		
9:
	uiStep :=  uiStep+1;
	state:=10;
	
10:(*Read *)
	bUp := FALSE;
	bDown:=FALSE;
	bDrain := FALSE;
	bN2  := FALSE;
	IF uiStep  <  5 THEN
		uiRemain :=rcp.uiRemain[ uiStep-1 ];
		uiCmd :=  rcp.uiCmd[ uiStep-1];
		IF uiRemain  > 0 THEN
			TotalStepRemain := TotalStepRemain -uiRemain;
			bUp 	:= GET_BIT_OF_INT(uiCmd , 0);
			bDown 	:= GET_BIT_OF_INT(uiCmd , 1);
			bN2 	:= GET_BIT_OF_INT(uiCmd , 2);
			bDrain 	:= GET_BIT_OF_INT(uiCmd ,3);
			state:=11;
		ELSE
			state:=9;
		END_IF;
	ELSIF uiStep  = 5 THEN
		IF LoopCount = 0 THEN
			state:=9;
		ELSE
			LoopCount := LoopCount -1;
			uiStep := 1;
			state:=9;
		END_IF;
	ELSIF uiStep  < 8 THEN
		uiRemain :=rcp.uiRemain[ uiStep-1 ];
		uiCmd :=  rcp.uiCmd[ uiStep-1];

		IF uiRemain  > 0 THEN
			TotalStepRemain := TotalStepRemain -uiRemain;
			bUp 	:= GET_BIT_OF_INT(uiCmd , 0);
			bDown 	:= GET_BIT_OF_INT(uiCmd , 1);
			bN2 	:= GET_BIT_OF_INT(uiCmd , 2);
			bDrain 	:= GET_BIT_OF_INT(uiCmd ,3);
			state:=11;
		ELSE
			state:=9;
		END_IF;
	ELSIF uiStep  = 8 THEN
			state:=20;
	END_IF;


11:
	TotalRemain := TotalStepRemain +uiRemain;
	IF  uiRemain <= 0 THEN
		state:=9;
	ELSIF NOT WaferIn AND SystemStart THEN
			state:=0;
	ELSIF BnMStart  AND NOT SystemStart THEN
		state:=0;
	ELSIF R_TRIG_1SEC.Q THEN
			uiRemain := uiRemain -1;
	END_IF;
	
20:
	bDone := TRUE;
	IF NOT WaferIn AND SystemStart THEN
			state:=0;
	ELSIF BnMStart  AND NOT SystemStart THEN
		state:=0;
	END_IF;


ELSE
	state :=0;
END_CASE;
END_FUNCTION_BLOCK
